// TwinCAT 3 PLC project Ligne
// ProgramVersion: 3.1.0.8
// libraries:
//   VisuElem3DPath, 3.5.4.0 (System)
//   VisuElemMeter, 3.5.4.0 (System)
//   VisuElems, 3.5.4.10 (System)
//   VisuElemsSpecialControls, 3.5.4.10 (System)
//   VisuElemsWinControls, 3.5.4.10 (System)
//   VisuElemTextEditor, 3.5.4.0 (System)
//   visuinputs, 3.5.4.0 (system)
//   VisuNativeControl, 3.5.4.0 (System)
//   Tc2_Standard, * (Beckhoff Automation GmbH)
//   Tc2_System, * (Beckhoff Automation GmbH)
//   Tc3_Interfaces, * (Beckhoff Automation GmbH)
//   Tc3_Module, * (Beckhoff Automation GmbH)
//   Maxon,1.0.0.0,Maxon Motor
//   Tc2_ControllerToolbox,3.4.1.0,Beckhoff Automation GmbH
//   Tc2_Utilities,3.3.8.0,Beckhoff Automation GmbH
// project tree:
//   DUTs/ FLAGS.TcDUT, FLOWMETER_CONTROL.TcDUT, FLOWMETER_SENSOR.TcDUT, FLOWMETER_VALUES.TcDUT, GAIN_SCHEDULED_PID.TcDUT, PRESSURE_SENSOR.TcDUT, PROG_STEPS.TcDUT, PUMP_PARAMS.TcDUT, SAFETY_IN.TcDUT, SAFETY_OUT.TcDUT
//   / GlobalTextList.TcGTLO, PlcTask.TcTTO, Visualization Manager.TcVMO (not stored)
//   GVLs/ Constant_Variables.TcGVL, Flag_Variables.TcGVL, IOs_Variables.TcGVL, PID_parameters.TcGVL
//   POUs/AIs/ AIS.TcPOU, ST45_TO_HMI.TcPOU
//   POUs/CONVOYER/ CONVEYOR.TcPOU, JIG.TcPOU
//   POUs/EAU/ VIDANGE_BALANCE_ST4.TcPOU, VIDANGE_BALANCE_ST5.TcPOU
//   POUs/EH/ EH_FLOMETER.TcPOU, EH_IEEE754_TO_REAL.TcPOU
//   POUs/Functions/ CONVERT_MASS_TO_FLOW.TcPOU, PRESSURE_REGULATOR.TcPOU
//   POUs/ GEMMA.TcPOU, MAIN.TcPOU
//   POUs/MAXON/ ST4_MOTOR.TcPOU, ST5_MOTOR.TcPOU, ST5_MOTOR_1.TcPOU
//   POUs/SAFETY/ SAFETY.TcPOU
//   POUs/STATIONS/ Q1.TcPOU, ST1_HT.TcPOU, ST2_ASPIRATION.TcPOU, ST3_ETANCHEITE.TcPOU, ST4_DEBIT_PETIT.TcPOU, ST5_GRAND_PETIT.TcPOU, ST7_SECHAGE.TcPOU, ST6_PMAX.TcPOU, ST8_IMPRESSION.TcPOU, ST9_DECHARGEMENT.TcPOU
//   POUs/WIKA/ WIKA_GET_VALUES.TcPOU
//   VISUs/ AIs.TcVIS, ST3.TcVIS, ST4.TcVIS, ST5.TcVIS, Visualization.TcVIS
// real-time tasks:
//   TASK PlcTask: cycle T#10ms, priority 20, ADS port 349
//   TASK Blinking: cycle T#450000us, priority 23, ADS port 351
//   TASK Slow_Tasks: cycle T#200000us, priority 22, ADS port 352
//   TASK TestOperator: cycle T#100000us, priority 21, ADS port 353
// I/O:
//   DEVICE Device 2 (EtherCAT), AmsNetId 10.10.10.31.3.1
//     Grande armoire [EK1100 EtherCAT Coupler (2A E-Bus)]
//       Term 51 (EL1002) [EL1002 2Ch. Dig. Input 24V, 3ms]
//       Term 52 (EL1002) [EL1002 2Ch. Dig. Input 24V, 3ms]
//       Term 53 (EL1002) [EL1002 2Ch. Dig. Input 24V, 3ms]
//       Term 54 (EL1002) [EL1002 2Ch. Dig. Input 24V, 3ms]
//       Term 55 (EL1002) [EL1002 2Ch. Dig. Input 24V, 3ms]
//       Term 56 (EL1002) [EL1002 2Ch. Dig. Input 24V, 3ms]
//       Term 57 (EL1002) [EL1002 2Ch. Dig. Input 24V, 3ms]
//       Term 58 (EL1002) [EL1002 2Ch. Dig. Input 24V, 3ms]
//       Term 59 (EL1002) [EL1002 2Ch. Dig. Input 24V, 3ms]
//       Term 60 (EL1002) [EL1002 2Ch. Dig. Input 24V, 3ms]
//       Term 61 (EL1002) [EL1002 2Ch. Dig. Input 24V, 3ms]
//       Term 62 (EL1002) [EL1002 2Ch. Dig. Input 24V, 3ms]
//       Term 63 (EL1002) [EL1002 2Ch. Dig. Input 24V, 3ms]
//       Term 64 (EL1002) [EL1002 2Ch. Dig. Input 24V, 3ms]
//       Term 65 (EL1002) [EL1002 2Ch. Dig. Input 24V, 3ms]
//       Term 66 (EL1002) [EL1002 2Ch. Dig. Input 24V, 3ms]
//       Term 67 (EL1002) [EL1002 2Ch. Dig. Input 24V, 3ms]
//       Term 68 (EL1002) [EL1002 2Ch. Dig. Input 24V, 3ms]
//       Term 32 (EL3064) [EL3064 4Ch. Ana. Input 0-10V]
//       Term 70 (EL1002) [EL1002 2Ch. Dig. Input 24V, 3ms]
//       Term 71 (EL9410) [EL9410 E-Bus Power Supplier  (Diagnostics)]
//       Term 72 (EL2002) [EL2002 2Ch. Dig. Output 24V, 0.5A]
//       Term 73 (EL2002) [EL2002 2Ch. Dig. Output 24V, 0.5A]
//       Term 74 (EL2002) [EL2002 2Ch. Dig. Output 24V, 0.5A]
//       Term 75 (EL2002) [EL2002 2Ch. Dig. Output 24V, 0.5A]
//       Term 76 (EL2002) [EL2002 2Ch. Dig. Output 24V, 0.5A]
//       Term 77 (EL2002) [EL2002 2Ch. Dig. Output 24V, 0.5A]
//       Term 78 (EL2002) [EL2002 2Ch. Dig. Output 24V, 0.5A]
//       Term 79 (EL2002) [EL2002 2Ch. Dig. Output 24V, 0.5A]
//       Term 80 (EL1512) [EL1512 2Ch. +/- Counter 24V, 1kHz]
//       Term 81 (EL2622) [EL2622 2Ch. Relay Output, NO (230V AC / 30V DC)]
//       Term 82 (EL2622) [EL2622 2Ch. Relay Output, NO (230V AC / 30V DC)]
//       Term 83 (EL2622) [EL2622 2Ch. Relay Output, NO (230V AC / 30V DC)]
//       Term 84 (EL2622) [EL2622 2Ch. Relay Output, NO (230V AC / 30V DC)]
//       Term 85 (EL2622) [EL2622 2Ch. Relay Output, NO (230V AC / 30V DC)]
//       Term 86 (EL2622) [EL2622 2Ch. Relay Output, NO (230V AC / 30V DC)]
//       Term 87 (EL3681) [EL3681 Digital multimeter terminal]
//       Term 88 (EL3681) [EL3681 Digital multimeter terminal]
//       Term 11 (EL2904) [EL2904, 4 Ch. Safety Output 24V, 0.5A, TwinSAFE]
//         modules: Module 1 (FSOES), Module 2 (DO)
//       Term 89 (EL6751) [EL6751 CANopen Master]
//       Term 90 (EL6751) [EL6751 CANopen Master]
//       Term 117 (EL9011) [EL9011 End Terminal]
//     Petite armoire [EK1100 EtherCAT Coupler (2A E-Bus)]
//       Term 92 (EL1002) [EL1002 2Ch. Dig. Input 24V, 3ms]
//       Term 93 (EL1002) [EL1002 2Ch. Dig. Input 24V, 3ms]
//       Term 94 (EL1002) [EL1002 2Ch. Dig. Input 24V, 3ms]
//       Term 95 (EL1002) [EL1002 2Ch. Dig. Input 24V, 3ms]
//       Term 96 (EL1002) [EL1002 2Ch. Dig. Input 24V, 3ms]
//       Term 97 (EL1002) [EL1002 2Ch. Dig. Input 24V, 3ms]
//       Term 98 (EL1002) [EL1002 2Ch. Dig. Input 24V, 3ms]
//       Term 99 (EL1002) [EL1002 2Ch. Dig. Input 24V, 3ms]
//       Term 100 (EL1002) [EL1002 2Ch. Dig. Input 24V, 3ms]
//       Term 101 (EL1002) [EL1002 2Ch. Dig. Input 24V, 3ms]
//       Term 102 (EL1002) [EL1002 2Ch. Dig. Input 24V, 3ms]
//       Term 103 (EL1002) [EL1002 2Ch. Dig. Input 24V, 3ms]
//       Term 104 (EL2002) [EL2002 2Ch. Dig. Output 24V, 0.5A]
//       Term 105 (EL2002) [EL2002 2Ch. Dig. Output 24V, 0.5A]
//       Term 106 (EL2002) [EL2002 2Ch. Dig. Output 24V, 0.5A]
//       Term 107 (EL2002) [EL2002 2Ch. Dig. Output 24V, 0.5A]
//       Term 149 (EL1008) [EL1008 8Ch. Dig. Input 24V, 3ms]
//       Term 150 (EL2008) [EL2008 8Ch. Dig. Output 24V, 0.5A]
//       Term 108 (EL3051) [EL3051 1Ch. Ana. Input 4-20mA]
//       Term 109 (EL9512) [EL9512 Power supply terminal 12V]
//       Term 110 (EL3356-0010) [EL3356-0010 1Ch. Ana. Input Resistor Bridge Terminal, 24bit, High Precision]
//       Term 111 (EL9512) [EL9512 Power supply terminal 12V]
//       Term 112 (EL3356-0010) [EL3356-0010 1Ch. Ana. Input Resistor Bridge Terminal, 24bit, High Precision]
//       Term 113 (EL6900) [EL6900, TwinSAFE PLC]
//       Term 114 (EL1904) [EL1904, 4 Ch. Safety Input 24V, TwinSAFE]
//         modules: Module 1 (FSOES)
//       Term 115 (EL1904) [EL1904, 4 Ch. Safety Input 24V, TwinSAFE]
//         modules: Module 1 (FSOES)
//       Term 116 (EL6731) [EL6731 PROFIBUS DP Master]
//       Term 118 (EL9011) [EL9011 End Terminal]
//     Box Etanchetie (EX260-SEC1) [EX260-SEC1 EtherCAT SI Unit (32DO_PNP) Rev1.2]
//     Box Debit (EX260-SEC1) [EX260-SEC1 EtherCAT SI Unit (32DO_PNP) Rev1.2]
//     Box Imprimante (EX260-SEC1) [EX260-SEC1 EtherCAT SI Unit (32DO_PNP) Rev1.2]
//   DEVICE Device 3 (EL6751), AmsNetId 10.10.10.31.4.1
//     Moteur Q1 (EPOS) (disabled)
//   DEVICE Device 4 (EL6751), AmsNetId 10.10.10.31.5.1
//     Moteur Q2 (EPOS) (disabled)
//   DEVICE Device 1 (EL6731), AmsNetId 10.10.10.31.2.1
//     Pressure Sensor 2P1 // Vendor: WIKA Revision: Rev 0.2
//     Pressure Sensor 4P2 // Vendor: WIKA Revision: Rev 0.2
//     Pressure Sensor 5P1 // Vendor: WIKA Revision: Rev 0.2
//     Pressure Sensor 5P2 // Vendor: WIKA Revision: Rev 0.2
//     Pressure Sensor 6P1 // Vendor: WIKA Revision: Rev 0.2
//     Pressure Sensor 4P1 // Vendor: WIKA Revision: Rev 0.2
// variable links:
//   Device 2 (EtherCAT) <-> Device 2 (EtherCAT)/Petite armoire/Term 113 (EL6900)
//     Grande armoire/Term 11 (EL2904)/Module 1 (FSOES)/RxPDO/FSOE <-> ConnectionInputs/Message_5 TxPDO
//     Grande armoire/Term 11 (EL2904)/Module 1 (FSOES)/TxPDO/FSOE <-> ConnectionOutputs/Message_5 RxPDO
//     Petite armoire/Term 114 (EL1904)/Module 1 (FSOES)/RxPDO/FSOE <-> ConnectionInputs/Message_24 TxPDO
//     Petite armoire/Term 114 (EL1904)/Module 1 (FSOES)/TxPDO/FSOE <-> ConnectionOutputs/Message_24 RxPDO
//     Petite armoire/Term 115 (EL1904)/Module 1 (FSOES)/TxPDO/FSOE <-> ConnectionOutputs/Message_4 RxPDO
//   Device 2 (EtherCAT) <-> Device 2 (EtherCAT)/Petite armoire/Term 115 (EL1904)
//     Petite armoire/Term 113 (EL6900)/ConnectionInputs/Message_4 TxPDO <-> Module 1 (FSOES)/RxPDO/FSOE
//   Ligne/Ligne Instance <-> Device 1 (EL6731)/Pressure Sensor 2P1
//     PlcTask Inputs/.ST2_2P1/VALUE <-> 8 Byte In, 3 Byte Out/Inputs/8 Byte In, 3 Byte Out_0_0
//   Ligne/Ligne Instance <-> Device 1 (EL6731)/Pressure Sensor 4P1
//     PlcTask Inputs/.ST4_4P1/VALUE <-> 8 Byte In, 3 Byte Out/Inputs/8 Byte In, 3 Byte Out_0_0
//   Ligne/Ligne Instance <-> Device 1 (EL6731)/Pressure Sensor 4P2
//     PlcTask Inputs/.ST4_4P2/VALUE <-> 8 Byte In, 3 Byte Out/Inputs/8 Byte In, 3 Byte Out_0_0
//   Ligne/Ligne Instance <-> Device 1 (EL6731)/Pressure Sensor 5P1
//     PlcTask Inputs/.ST5_5P1/VALUE <-> 8 Byte In, 3 Byte Out/Inputs/8 Byte In, 3 Byte Out_0_0
//   Ligne/Ligne Instance <-> Device 1 (EL6731)/Pressure Sensor 5P2
//     PlcTask Inputs/.ST5_5P2/VALUE <-> 8 Byte In, 3 Byte Out/Inputs/8 Byte In, 3 Byte Out_0_0
//   Ligne/Ligne Instance <-> Device 1 (EL6731)/Pressure Sensor 6P1
//     PlcTask Inputs/.ST6_6P1/VALUE <-> 8 Byte In, 3 Byte Out/Inputs/8 Byte In, 3 Byte Out_0_0
//   Ligne/Ligne Instance <-> Device 2 (EtherCAT)/Box Debit (EX260-SEC1)
//     PlcTask Outputs/.ST4_4V1 <-> Byte 0/Output
//     PlcTask Outputs/.ST5_5V2 <-> Byte 1/Output
//     PlcTask Outputs/.ST6_6V4 <-> Byte 2/Output
//     PlcTask Outputs/.ST4_4V2 <-> Byte 0/Output @bit 1
//     PlcTask Outputs/.ST4_4V3 <-> Byte 0/Output @bit 2
//     PlcTask Outputs/.ST4_4V4 <-> Byte 0/Output @bit 3
//     PlcTask Outputs/.ST4_4V5 <-> Byte 0/Output @bit 4
//     PlcTask Outputs/.ST4_4V6 <-> Byte 0/Output @bit 5
//     PlcTask Outputs/.ST4_4V7 <-> Byte 0/Output @bit 6
//     PlcTask Outputs/.ST5_5V1 <-> Byte 0/Output @bit 7
//     PlcTask Outputs/.ST5_5V3 <-> Byte 1/Output @bit 1
//     PlcTask Outputs/.ST5_5V4 <-> Byte 1/Output @bit 2
//     PlcTask Outputs/.ST5_5V5 <-> Byte 1/Output @bit 3
//     PlcTask Outputs/.ST5_5V6 <-> Byte 1/Output @bit 4
//     PlcTask Outputs/.ST6_6V1 <-> Byte 1/Output @bit 5
//     PlcTask Outputs/.ST6_6V2 <-> Byte 1/Output @bit 6
//     PlcTask Outputs/.ST6_6V3 <-> Byte 1/Output @bit 7
//     PlcTask Outputs/.ST6_6V5 <-> Byte 2/Output @bit 1
//     PlcTask Outputs/.ST6_6V6 <-> Byte 2/Output @bit 2
//     PlcTask Outputs/.ST6_6V7 <-> Byte 2/Output @bit 3
//   Ligne/Ligne Instance <-> Device 2 (EtherCAT)/Box Etanchetie (EX260-SEC1)
//     PlcTask Outputs/.ST10_10V1 <-> Byte 0/Output
//     PlcTask Outputs/.ST2_2V2 <-> Byte 1/Output
//     PlcTask Outputs/.ST3_3V3 <-> Byte 2/Output
//     PlcTask Outputs/.ST10_10V2 <-> Byte 0/Output @bit 1
//     PlcTask Outputs/.ST1_1V1 <-> Byte 0/Output @bit 2
//     PlcTask Outputs/.ST1_1V2 <-> Byte 0/Output @bit 3
//     PlcTask Outputs/.ST1_1V3 <-> Byte 0/Output @bit 4
//     PlcTask Outputs/.ST1_1V4 <-> Byte 0/Output @bit 5
//     PlcTask Outputs/.ST1_1V5 <-> Byte 0/Output @bit 6
//     PlcTask Outputs/.ST2_2V1 <-> Byte 0/Output @bit 7
//     PlcTask Outputs/.ST2_2V3 <-> Byte 1/Output @bit 1
//     PlcTask Outputs/.ST2_2V4 <-> Byte 1/Output @bit 2
//     PlcTask Outputs/.ST2_2V5 <-> Byte 1/Output @bit 3
//     PlcTask Outputs/.ST2_2V6 <-> Byte 1/Output @bit 4
//     PlcTask Outputs/.ST2_2V7 <-> Byte 1/Output @bit 5
//     PlcTask Outputs/.ST3_3V1 <-> Byte 1/Output @bit 6
//     PlcTask Outputs/.ST3_3V2 <-> Byte 1/Output @bit 7
//     PlcTask Outputs/.ST3_3V4 <-> Byte 2/Output @bit 1
//     PlcTask Outputs/.ST3_3V5 <-> Byte 2/Output @bit 2
//     PlcTask Outputs/.ST3_3V7 <-> Byte 2/Output @bit 3
//   Ligne/Ligne Instance <-> Device 2 (EtherCAT)/Box Imprimante (EX260-SEC1)
//     PlcTask Outputs/.ST7_7V1 <-> Byte 0/Output @bit 1
//     PlcTask Outputs/.ST7_7V2 <-> Byte 0/Output @bit 2
//     PlcTask Outputs/.ST7_7V3 <-> Byte 0/Output @bit 3
//     PlcTask Outputs/.ST7_7V4 <-> Byte 0/Output @bit 4
//     PlcTask Outputs/.ST7_7V5 <-> Byte 0/Output @bit 5
//     PlcTask Outputs/.ST7_7V6 <-> Byte 0/Output @bit 6
//     PlcTask Outputs/.ST7_7V7 <-> Byte 0/Output @bit 7
//     PlcTask Outputs/.ST8_8V2 <-> Byte 1/Output @bit 1
//     PlcTask Outputs/.ST8_8V3 <-> Byte 1/Output @bit 2
//     PlcTask Outputs/.ST8_8V4 <-> Byte 1/Output @bit 3
//     PlcTask Outputs/.ST9_9V1 <-> Byte 1/Output @bit 4
//     PlcTask Outputs/.ST9_9V2 <-> Byte 1/Output @bit 5
//     PlcTask Outputs/.ST9_9V3 <-> Byte 1/Output @bit 6
//     PlcTask Outputs/.ST9_9V6 <-> Byte 2/Output @bit 3
//     PlcTask Outputs/.ST9_9V7 <-> Byte 2/Output @bit 4
//     PlcTask Outputs/.ST7_RESERVE <-> Byte 0/Output
//     PlcTask Outputs/.ST8_8V1 <-> Byte 1/Output
//     PlcTask Outputs/.ST9_9V4A <-> Byte 1/Output @bit 7
//     PlcTask Outputs/.ST9_9V5A <-> Byte 2/Output @bit 1
//     PlcTask Outputs/.ST9_9V4B <-> Byte 2/Output
//     PlcTask Outputs/.ST9_9V5B <-> Byte 2/Output @bit 2
//   Ligne/Ligne Instance <-> Device 2 (EtherCAT)/Grande armoire/Term 32 (EL3064)
//     PlcTask Inputs/.ST3_3P2 <-> AI Standard Channel 4/Value
//     PlcTask Inputs/.ST5_Niveau_Reservoir <-> AI Standard Channel 3/Value
//   Ligne/Ligne Instance <-> Device 2 (EtherCAT)/Grande armoire/Term 51 (EL1002)
//     PlcTask Inputs/.ST4_4B1 <-> Channel 1/4B1
//     PlcTask Inputs/.ST4_4B2 <-> Channel 2/4B2
//   Ligne/Ligne Instance <-> Device 2 (EtherCAT)/Grande armoire/Term 52 (EL1002)
//     PlcTask Inputs/.ST4_4B4 <-> Channel 1/4B4
//     PlcTask Inputs/.ST4_4B5 <-> Channel 2/4B5
//   Ligne/Ligne Instance <-> Device 2 (EtherCAT)/Grande armoire/Term 53 (EL1002)
//     PlcTask Inputs/.ST4_4B6 <-> Channel 1/4B6
//     PlcTask Inputs/.ST4_4B7 <-> Channel 2/4B7
//   Ligne/Ligne Instance <-> Device 2 (EtherCAT)/Grande armoire/Term 54 (EL1002)
//     PlcTask Inputs/.ST5_5B1 <-> Channel 1/5B1
//     PlcTask Inputs/.ST5_5B2 <-> Channel 2/5B2
//   Ligne/Ligne Instance <-> Device 2 (EtherCAT)/Grande armoire/Term 55 (EL1002)
//     PlcTask Inputs/.ST5_5B4 <-> Channel 1/5B4
//     PlcTask Inputs/.ST5_5B5 <-> Channel 2/5B5
//   Ligne/Ligne Instance <-> Device 2 (EtherCAT)/Grande armoire/Term 56 (EL1002)
//     PlcTask Inputs/.ST5_5B6 <-> Channel 1/5B6
//   Ligne/Ligne Instance <-> Device 2 (EtherCAT)/Grande armoire/Term 57 (EL1002)
//     PlcTask Inputs/.ST6_6B1 <-> Channel 1/6B1
//     PlcTask Inputs/.ST6_6B2 <-> Channel 2/6B2
//   Ligne/Ligne Instance <-> Device 2 (EtherCAT)/Grande armoire/Term 58 (EL1002)
//     PlcTask Inputs/.ST6_6B4 <-> Channel 1/6B4
//     PlcTask Inputs/.ST6_6B5 <-> Channel 2/6B5
//   Ligne/Ligne Instance <-> Device 2 (EtherCAT)/Grande armoire/Term 59 (EL1002)
//     PlcTask Inputs/.ST6_6B6 <-> Channel 1/6B6
//     PlcTask Inputs/.ST6_6B7 <-> Channel 2/6B7
//   Ligne/Ligne Instance <-> Device 2 (EtherCAT)/Grande armoire/Term 60 (EL1002)
//     PlcTask Inputs/.ST7_7B1 <-> Channel 1/7B1
//     PlcTask Inputs/.ST7_7B2 <-> Channel 2/7B2
//   Ligne/Ligne Instance <-> Device 2 (EtherCAT)/Grande armoire/Term 61 (EL1002)
//     PlcTask Inputs/.ST7_7B4 <-> Channel 1/7B4
//     PlcTask Inputs/.ST7_7B5 <-> Channel 2/7B5
//   Ligne/Ligne Instance <-> Device 2 (EtherCAT)/Grande armoire/Term 62 (EL1002)
//     PlcTask Inputs/.ST7_7B6 <-> Channel 1/7B6
//     PlcTask Inputs/.ST7_7B7 <-> Channel 2/7B7
//   Ligne/Ligne Instance <-> Device 2 (EtherCAT)/Grande armoire/Term 63 (EL1002)
//     PlcTask Inputs/.ST8_8B1 <-> Channel 1/8B1
//     PlcTask Inputs/.ST8_8B2 <-> Channel 2/8B2
//   Ligne/Ligne Instance <-> Device 2 (EtherCAT)/Grande armoire/Term 64 (EL1002)
//     PlcTask Inputs/.ST9_9B1 <-> Channel 1/9B1
//     PlcTask Inputs/.ST9_9B2 <-> Channel 2/9B2
//   Ligne/Ligne Instance <-> Device 2 (EtherCAT)/Grande armoire/Term 65 (EL1002)
//     PlcTask Inputs/.ST9_9B4 <-> Channel 1/9B4
//     PlcTask Inputs/.ST9_9B41 <-> Channel 2/9B4.1
//   Ligne/Ligne Instance <-> Device 2 (EtherCAT)/Grande armoire/Term 66 (EL1002)
//     PlcTask Inputs/.ST9_9B5 <-> Channel 1/9B5
//     PlcTask Inputs/.ST9_9B51 <-> Channel 2/9B5.1
//   Ligne/Ligne Instance <-> Device 2 (EtherCAT)/Grande armoire/Term 67 (EL1002)
//     PlcTask Inputs/.ST9_9B6 <-> Channel 1/9B6
//     PlcTask Inputs/.ST9_9B7 <-> Channel 2/9B7
//   Ligne/Ligne Instance <-> Device 2 (EtherCAT)/Grande armoire/Term 68 (EL1002)
//     PlcTask Inputs/.ST9_9B61 <-> Channel 2/9B6.1
//   Ligne/Ligne Instance <-> Device 2 (EtherCAT)/Grande armoire/Term 72 (EL2002)
//     PlcTask Outputs/.ST4_4V10 <-> Channel 1/4V10
//     PlcTask Outputs/.ST4_4V12 <-> Channel 2/4V12
//   Ligne/Ligne Instance <-> Device 2 (EtherCAT)/Grande armoire/Term 73 (EL2002)
//     PlcTask Outputs/.ST4_4V13 <-> Channel 1/4V13
//   Ligne/Ligne Instance <-> Device 2 (EtherCAT)/Grande armoire/Term 74 (EL2002)
//     PlcTask Outputs/.ST5_5V10 <-> Channel 1/5V10
//     PlcTask Outputs/.ST5_5V12 <-> Channel 2/5V12
//   Ligne/Ligne Instance <-> Device 2 (EtherCAT)/Grande armoire/Term 75 (EL2002)
//     PlcTask Outputs/.ST5_5V13 <-> Channel 1/5V13
//     PlcTask Outputs/.ST5_5V14 <-> Channel 2/5V14
//   Ligne/Ligne Instance <-> Device 2 (EtherCAT)/Grande armoire/Term 76 (EL2002)
//     PlcTask Outputs/.ST5_5V15 <-> Channel 1/5V15
//     PlcTask Outputs/.ST5_5V16 <-> Channel 2/5V16
//   Ligne/Ligne Instance <-> Device 2 (EtherCAT)/Grande armoire/Term 77 (EL2002)
//     PlcTask Outputs/.ST6_6V10 <-> Channel 1/6V10
//     PlcTask Outputs/.ST6_6V11 <-> Channel 2/6V11
//   Ligne/Ligne Instance <-> Device 2 (EtherCAT)/Grande armoire/Term 78 (EL2002)
//     PlcTask Outputs/.GEN_CONVOYEUR <-> Channel 1/K2
//   Ligne/Ligne Instance <-> Device 2 (EtherCAT)/Grande armoire/Term 79 (EL2002)
//     PlcTask Outputs/.ST7_7V10 <-> Channel 1/7V10
//   Ligne/Ligne Instance <-> Device 2 (EtherCAT)/Grande armoire/Term 81 (EL2622)
//     PlcTask Outputs/.ST2_POWER <-> Channel 1/2M1L
//     PlcTask Outputs/.ST2_POWER <-> Channel 2/2M1N
//   Ligne/Ligne Instance <-> Device 2 (EtherCAT)/Grande armoire/Term 82 (EL2622)
//     PlcTask Outputs/.ST4_POWER <-> Channel 1/4M1L
//     PlcTask Outputs/.ST4_POWER <-> Channel 2/4M1N
//   Ligne/Ligne Instance <-> Device 2 (EtherCAT)/Grande armoire/Term 83 (EL2622)
//     PlcTask Outputs/.ST5_POWER <-> Channel 1/5M1L
//     PlcTask Outputs/.ST5_POWER <-> Channel 2/5M1N
//   Ligne/Ligne Instance <-> Device 2 (EtherCAT)/Grande armoire/Term 84 (EL2622)
//     PlcTask Outputs/.ST6_POWER <-> Channel 1/6M1L
//     PlcTask Outputs/.ST6_POWER <-> Channel 2/6M1N
//   Ligne/Ligne Instance <-> Device 2 (EtherCAT)/Grande armoire/Term 85 (EL2622)
//     PlcTask Outputs/.ST7_POWER <-> Channel 1/7M1L
//     PlcTask Outputs/.ST7_POWER <-> Channel 2/7M1N
//   Ligne/Ligne Instance <-> Device 2 (EtherCAT)/Grande armoire/Term 86 (EL2622)
//     PlcTask Outputs/.ST4_VIDANGE <-> Channel 1/4M2
//     PlcTask Outputs/.ST5_VIDANGE <-> Channel 2/5M2
//   Ligne/Ligne Instance <-> Device 2 (EtherCAT)/Grande armoire/Term 87 (EL3681)
//     PlcTask Inputs/.ST4_Multimeter_value <-> SAI Inputs/Value
//     PlcTask Outputs/.ST4_Multimeter_mode <-> SAI Range/Control/Mode
//     PlcTask Outputs/.ST4_Multimeter_range <-> SAI Range/Control/Range
//   Ligne/Ligne Instance <-> Device 2 (EtherCAT)/Grande armoire/Term 88 (EL3681)
//     PlcTask Inputs/.ST5_Multimeter_value <-> SAI Inputs/Value
//     PlcTask Outputs/.ST5_Multimeter_mode <-> SAI Range/Control/Mode
//     PlcTask Outputs/.ST5_Multimeter_range <-> SAI Range/Control/Range
//   Ligne/Ligne Instance <-> Device 2 (EtherCAT)/Petite armoire/Term 100 (EL1002)
//     PlcTask Inputs/.GEN_PRESENCE_POMPE <-> Channel 1/Présence pompe
//   Ligne/Ligne Instance <-> Device 2 (EtherCAT)/Petite armoire/Term 101 (EL1002)
//     PlcTask Inputs/.ST4_DIGMESA <-> Channel 1/Input
//   Ligne/Ligne Instance <-> Device 2 (EtherCAT)/Petite armoire/Term 102 (EL1002)
//     PlcTask Inputs/.ST10_OPERATEUR1_START <-> Channel 1/S1
//     PlcTask Inputs/.ST10_OPERATEUR2_START <-> Channel 2/S2
//   Ligne/Ligne Instance <-> Device 2 (EtherCAT)/Petite armoire/Term 103 (EL1002)
//     PlcTask Inputs/.ST10_10B1 <-> Channel 1/10B1
//     PlcTask Inputs/.ST10_10B2 <-> Channel 2/10B2
//   Ligne/Ligne Instance <-> Device 2 (EtherCAT)/Petite armoire/Term 104 (EL2002)
//     PlcTask Outputs/.ST3_3V10 <-> Channel 1/3V10
//     PlcTask Outputs/.ST3_3V11 <-> Channel 2/3V11
//   Ligne/Ligne Instance <-> Device 2 (EtherCAT)/Petite armoire/Term 105 (EL2002)
//     PlcTask Outputs/.ST2_2V8 <-> Channel 2/2V8
//     PlcTask Outputs/.ST3_3V12 <-> Channel 1/3V12
//   Ligne/Ligne Instance <-> Device 2 (EtherCAT)/Petite armoire/Term 106 (EL2002)
//     PlcTask Outputs/.GEN_1V1 <-> Channel 1/0V1
//   Ligne/Ligne Instance <-> Device 2 (EtherCAT)/Petite armoire/Term 108 (EL3051)
//     PlcTask Inputs/.ST3_3P1 <-> AI Standard/3P1
//   Ligne/Ligne Instance <-> Device 2 (EtherCAT)/Petite armoire/Term 110 (EL3356-0010)
//     PlcTask Inputs/.ST4_POIDS <-> RMB Value (Real)/4U1
//   Ligne/Ligne Instance <-> Device 2 (EtherCAT)/Petite armoire/Term 112 (EL3356-0010)
//     PlcTask Inputs/.ST5_POIDS <-> RMB Value (Real)/5U1
//   Ligne/Ligne Instance <-> Device 2 (EtherCAT)/Petite armoire/Term 113 (EL6900)
//     PlcTask Inputs/.SAFETY_IN/NOT_AUS_State <-> Function Block Info Data/TwinSafeGroup2.Network1.FBEstop1 Info Data/State
//     PlcTask Outputs/.SAFETY_OUT/NOT_AUS_ErrAck <-> StandardOutputs/Standard In Var 9
//     PlcTask Outputs/.SAFETY_OUT/NOT_AUS_RESET <-> StandardOutputs/Standard In Var 10
//     PlcTask Outputs/.SAFETY_OUT/NOT_AUS_RUN <-> StandardOutputs/Standard In Var 8
//   Ligne/Ligne Instance <-> Device 2 (EtherCAT)/Petite armoire/Term 149 (EL1008)
//     PlcTask Inputs/.ST1_HT_CTRLOUT <-> Channel 1/HT_CTRLout
//     PlcTask Inputs/.ST1_HT_EOT <-> Channel 2/HT_EOT
//     PlcTask Inputs/.ST1_HT_ERROR <-> Channel 5/ERROR
//     PlcTask Inputs/.ST1_HT_FAIL <-> Channel 4/HT_FAIL
//     PlcTask Inputs/.ST1_HT_PASS <-> Channel 3/HT_PASS
//   Ligne/Ligne Instance <-> Device 2 (EtherCAT)/Petite armoire/Term 150 (EL2008)
//     PlcTask Outputs/.ST1_HT_CTRLIN <-> Channel 1/HT_CTRLIN
//     PlcTask Outputs/.ST1_HT_MES_DCH <-> Channel 6/HT_MES_DCH
//     PlcTask Outputs/.ST1_HT_N0 <-> Channel 3/HT_N0
//     PlcTask Outputs/.ST1_HT_N1 <-> Channel 4/HT_N1
//     PlcTask Outputs/.ST1_HT_N2 <-> Channel 5/HT_N2
//     PlcTask Outputs/.ST1_HT_TYPW <-> Channel 2/HT_TYPE
//   Ligne/Ligne Instance <-> Device 2 (EtherCAT)/Petite armoire/Term 92 (EL1002)
//     PlcTask Inputs/.ST1_1B1 <-> Channel 1/1B1
//     PlcTask Inputs/.ST1_1B2 <-> Channel 2/1B2
//   Ligne/Ligne Instance <-> Device 2 (EtherCAT)/Petite armoire/Term 93 (EL1002)
//     PlcTask Inputs/.ST1_1B4 <-> Channel 1/1B4
//     PlcTask Inputs/.ST1_1B5 <-> Channel 2/1B5
//   Ligne/Ligne Instance <-> Device 2 (EtherCAT)/Petite armoire/Term 94 (EL1002)
//     PlcTask Inputs/.ST2_2B1 <-> Channel 1/2B1
//     PlcTask Inputs/.ST2_2B2 <-> Channel 2/2B2
//   Ligne/Ligne Instance <-> Device 2 (EtherCAT)/Petite armoire/Term 95 (EL1002)
//     PlcTask Inputs/.ST2_2B4 <-> Channel 1/2B4
//     PlcTask Inputs/.ST2_2B5 <-> Channel 2/2B5
//   Ligne/Ligne Instance <-> Device 2 (EtherCAT)/Petite armoire/Term 96 (EL1002)
//     PlcTask Inputs/.ST2_2B6 <-> Channel 1/2B6
//     PlcTask Inputs/.ST2_2B7 <-> Channel 2/2B7
//   Ligne/Ligne Instance <-> Device 2 (EtherCAT)/Petite armoire/Term 97 (EL1002)
//     PlcTask Inputs/.ST3_3B1 <-> Channel 1/3B1
//     PlcTask Inputs/.ST3_3B2 <-> Channel 2/3B2
//   Ligne/Ligne Instance <-> Device 2 (EtherCAT)/Petite armoire/Term 98 (EL1002)
//     PlcTask Inputs/.ST3_3B4 <-> Channel 1/3B4
//     PlcTask Inputs/.ST3_3B5 <-> Channel 2/3B5
//   Ligne/Ligne Instance <-> Device 2 (EtherCAT)/Petite armoire/Term 99 (EL1002)
//     PlcTask Inputs/.GEN_0B1 <-> Channel 2/0B1
//     PlcTask Inputs/.ST3_3B7 <-> Channel 1/3B7

CONFIGURATION Ligne
    RESOURCE PLC ON TwinCAT3
        TASK PlcTask(INTERVAL := T#10ms, PRIORITY := 20);
        PROGRAM MAIN WITH PlcTask : MAIN;
    END_RESOURCE
END_CONFIGURATION

// ---- DUTs/FLAGS.TcDUT
TYPE FLAGS :
STRUCT

	INIT_OK:BOOL;
	SAFETY_OK:BOOL;
	MANUAL:BOOL;
	AUTO:BOOL;
	
	DEBUG_OPERATOR:BOOL;
	
	ST1_JIG_STATUS: BOOL;
	ST1_RELEASE_CARRIER:BOOL;
	ST2_JIG_STATUS: BOOL;
	ST2_RELEASE_CARRIER:BOOL;
	ST3_JIG_STATUS: BOOL;
	ST3_RELEASE_CARRIER:BOOL;
	ST4_JIG_STATUS: BOOL;
	ST4_RELEASE_CARRIER:BOOL;
	ST5_JIG_STATUS: BOOL;
	ST5_RELEASE_CARRIER:BOOL;
	ST6_JIG_STATUS: BOOL;
	ST6_RELEASE_CARRIER:BOOL;
	ST7_JIG_STATUS: BOOL;
	ST7_RELEASE_CARRIER:BOOL;
	ST8_JIG_STATUS: BOOL;
	ST8_RELEASE_CARRIER:BOOL;
	ST9_JIG_STATUS: BOOL;
	ST9_RELEASE_CARRIER:BOOL;

	
	DOORS_OPEN:BOOL;
	F2_END:BOOL;
	GEMMA: STRING;
	
	MOTOR_ST4_INIT_OK:BOOL;
	MOTOR_ST4_POSITION:DINT;
	MOTOR_ST4_ACTUAL_POSITION:DINT;
	MOTOR_ST5_INIT_OK:BOOL;
	MOTOR_ST5_POSITION:DINT;
	MOTOR_ST5_ACTUAL_POSITION:DINT;



END_STRUCT
END_TYPE

// ---- DUTs/FLOWMETER_CONTROL.TcDUT
TYPE FLOWMETER_CONTROL :
STRUCT

	SET_TOT: USINT;
	SET_MODE: USINT;

END_STRUCT
END_TYPE

// ---- DUTs/FLOWMETER_SENSOR.TcDUT

(************************************************************************************************
*
*Variables structure for E&H flowmeter PROMAS 83A
*
***********************************************************************************************)


TYPE FLOWMETER_SENSOR :
STRUCT

	A1 :ARRAY[0..4] OF USINT;
	A2 :ARRAY[0..4] OF USINT;
	A3 :ARRAY[0..4] OF USINT;
	A4 :ARRAY[0..4] OF USINT;
	A5 :ARRAY[0..4] OF USINT;
	A6 :ARRAY[0..4] OF USINT;
	TOT :ARRAY[0..4] OF USINT;

END_STRUCT
END_TYPE

// ---- DUTs/FLOWMETER_VALUES.TcDUT
TYPE FLOWMETER_VALUES :
STRUCT
	MassFlow:REAL;
	VolumeFlow:REAL;
	CorrectedVolueFLow:REAL;
	Density:REAL;
	ReferenceDensity:REAL;
	Temperature:REAL;
	TotalMass:REAL;
END_STRUCT
END_TYPE

// ---- DUTs/GAIN_SCHEDULED_PID.TcDUT
TYPE GAIN_SCHEDULED_PID :
STRUCT
	q			:REAL; 	(*gain scheduled parameter for which this PID is optimized*)
	Kp			:REAL;	(*constant for proportional part of the PID*)
	Ki			:REAL;	(*constant for integral part of the PID*)
	Kd			:REAL;	(*constant for derivative part of the PID*)
END_STRUCT
END_TYPE

// ---- DUTs/PRESSURE_SENSOR.TcDUT

(************************************************************************************************
*
*Variables structure for WIKA pressure sensor
*
***********************************************************************************************)

TYPE PRESSURE_SENSOR :
STRUCT

	VALUE :ARRAY [0..7] OF USINT;

END_STRUCT
END_TYPE

// ---- DUTs/PROG_STEPS.TcDUT
TYPE PROG_STEPS :
STRUCT

	ST1:INT;
	ST2:INT;
	ST3:INT;
	ST4:INT;
	ST5:INT;
	ST6:INT;
	ST7:INT;
	ST8:INT;
	ST9:INT;


END_STRUCT
END_TYPE

// ---- DUTs/PUMP_PARAMS.TcDUT
TYPE PUMP_PARAMS :
STRUCT
	
(* Général *******************************************************************************************************************)
	GEN_GRAND_DEBIT					:BOOL:=FALSE;		(*FALSE / ST4 petit débit     TRUE / ST5 grand débit*)
	GEN_BYPASS						:BOOL:=FALSE;		(*FALSE / N'utilise pas le contrôle du bypass      TRUE / Utilise le contrôle du by-pass*)
		
	
(* Station 1 Haute tension ***************************************************************************************************)
	ST1_HT_NO_PROG					:INT:=1;			(*Numéro de programme de l'appareil de test HT*)

(* Station 2 aspiration ******************************************************************************************************)
	ST2_CONTRE_PRESSION				:BOOL:=0;			(*Contre pression d'air TRUE: avec contre pression FALSE: sans contre pression*)
	ST2_TEMPS_POMPAGE				:TIME:= T#10S;		(*Temps d'amorcage *)
	ST2_TEMPS_MESURE				:TIME:= T#5S;		(*Temps de mesure *)
	ST2_TEMPS_MESURE_PERTE_PRESSION	:TIME:= T#2S;		(*Temps de mesure perte pression - PAS PROGRAMME *)
		
(* Station 3 étanchéité ******************************************************************************************************)
	ST3_TEMPS_MISE_SOUS_PRESSION	:TIME:= T#5S;		(*Temps de mise sous pression*)
	ST3_TEMPS_STABILISATION			:TIME:= T#10S;		(*Temps de stabilisation de la pression*)
	ST3_TEMPS_MESURE				:TIME:= T#15S;		(*Temps de mesure de la chutte de	 pression*)
	

(* Station 4-5 Débit *****************************************************************************************************)
	ST45_TEMPS_POMPAGE				:TIME:= T#10S;		(*Temps amorcage de la pompe *)
	ST45_TEMPS_MESURE_DEBIT_MAX		:TIME:= T#10S;		(*Temps de mesure de Qmax*)
	ST45_TEMPS_REGLAGE_PRESSION		:TIME:= T#30S;		(*Temps de réglage de la pression *)
	ST45_TEMPS_MESURE_DEBIT			:TIME:= T#10S;		(*Temps de mesure de Qtravail *)
	ST45_PRESSION_CONSIGNE			:REAL:= 7.0;		(*Presssion de consigne pour le débit de travail*)

(* Station 6 Pmax ************************************************************************************************************)	
	ST6_TEMPS_POMPAGE				:TIME:= T#10S;		(*Temps amorcage de la pompe *)
	ST6_TEMPS_MESURE				:TIME:= T#5S;		(*Temps de mesure de Pmax *)
	ST6_TEMPS_MESURE_PERTE_PRESSION	:TIME:= T#1S;		(*Temps de mesure perte de pression max - PAS PROGRAMME *)
	
(* Station 7 Sechage *********************************************************************************************************)
	ST7_TEMPS_SECHAGE				:TIME:= T#2S;		(*Temps séchage pompe station 7 *)
	
(* Station 9 Déchargement*****************************************************************************************************)
	ST9_BOBINE_A_FIL				:BOOL:=TRUE;		(*Si bobine à fil, utilise de vérin de débloquage des fils *)



END_STRUCT
END_TYPE

// ---- DUTs/SAFETY_IN.TcDUT
TYPE SAFETY_IN :
STRUCT

	NOT_AUS_State:USINT;

END_STRUCT
END_TYPE

// ---- DUTs/SAFETY_OUT.TcDUT
TYPE SAFETY_OUT :
STRUCT


	NOT_AUS_RUN:BOOL;
	NOT_AUS_ErrAck:BOOL;
	NOT_AUS_RESET:BOOL;

END_STRUCT
END_TYPE

// ---- GVLs/Constant_Variables.TcGVL
{attribute 'Tc2GvlVarNames'}
VAR_GLOBAL
	(********************
	*
	* Times
	*  
	************************)
	CARRIER_RELEASE_DELAY						:TIME:= T#600MS;			(*Temps de rentrée du vérin de blocage des vérins*)
	PULSE_RELEASE_JIG_OP						:TIME:= T#250MS;		(*Duration of the pulse to release a carrier on the Operators jig*)
	DELAY_EJECT_CARRIERS						:TIME:= T#5S;			(*Time for release all the carriers present in the tunel during the initialisation *)
	DELAY_START_AIR								:TIME:= T#2S;			(*Time to let air starting before starting convoyer *)

	TEMPS_VIDANGE_POMPE							:TIME:= T#5S;			(*Temps durant lequel on pompe de l'air pour vidanger la pompe*)
	TEMPS_VIDANGE_RESERVOIR						:TIME:= T#30S;			(*Temps durant lequel on continue de vider le réservoir d'eau pour être sur qu'il est vide*)
	
	TEMPS_SORTIE_VERIN							:TIME:= T#3S;			(*Temps durant lequel on pompe de l'air pour vidanger la pompe*)
	TEMPS_RENTREE_VERIN							:TIME:= T#1S;			(*Temps laissé au vérin pour rentrer avant que la palette soit libérée*)
	TEMPS_CHANGEMENT_PRESSION					:TIME:= T#4S;			(*Temps pour la mise sous pression du débit de travail avant réglage*)

	(********************
	*
	* Motor
	*
	************************)
	MOTOR_ST4_ADDRESS							:STRING:= '10.10.10.31.4.1';	(*Adresse moteur ST4*)
	MOTOR_ST5_ADDRESS							:STRING:= '10.10.10.31.5.1';	(*Adresse moteur ST5*)
	MOTOR_ST4_INITIAL_POS						:DINT:=25000;					(*Initial position of the motor*)
	MOTOR_ST4_POSITION_MAX						:DINT:=35000;					(*Butée soft du moteur*)
	MOTOR_ST5_INITIAL_POS						:DINT:=25000;					(*Initial position of the motor*)
	MOTOR_ST5_POSITION_MAX						:DINT:=35000;					(*Butée soft du moteur*)
	
	RESERVOIR_EAU_MAX							:INT:=5000;						(*Niveau haut du réservoir d'eau*)
	RESERVOIR_EAU_MIN							:INT:=14000;					(*Niveau bas du réservoir d'eau*)
	
	(********************
	*
	* Weigthing
	*
	************************)
	
	BALANCE_POIDS_LIMITE								:INT:=2000;

END_VAR

VAR_GLOBAL

	(********************
	*
	* Config
	*
	************************)

	PUMP_PARAMS 									: PUMP_PARAMS;		(*Paramètre de test qu viennent depuis Labview*)

	(********************
	*
	* Activation des Posages
	*
	************************)
	ST1_JIG_DISABLED							:BOOL:=FALSE;			(*Désactive le posage*)
	ST2_JIG_DISABLED							:BOOL:=FALSE;			(*Désactive le posage*)
	ST3_JIG_DISABLED							:BOOL:=FALSE;			(*Désactive le posage*)
	ST4_5_JIG_DISABLED							:BOOL:=FALSE;			(*Désactive les posages ST4 et ST5*)
	ST6_JIG_DISABLED							:BOOL:=FALSE;			(*Désactive le posage*)
	ST7_JIG_DISABLED							:BOOL:=FALSE;			(*Désactive le posage*)
	ST8_JIG_DISABLED							:BOOL:=FALSE;			(*Désactive le posage*)
	ST9_JIG_DISABLED							:BOOL:=FALSE;			(*Désactive le posage*)
	ST4_JIG_DISABLED							:BOOL;					(*via la variable GRAND_DEBIT*)
	ST5_JIG_DISABLED							:BOOL;					(*via la variable GRAND_DEBIT*)

END_VAR

// ---- GVLs/Flag_Variables.TcGVL
{attribute 'Tc2GvlVarNames'}
VAR_GLOBAL


	FLAGS 				AT%M*: FLAGS;


	SAFETY_IN 			AT%I*: SAFETY_IN;
	SAFETY_OUT 			AT%Q*: SAFETY_OUT;

	(*Visualisation des débits ST4*)
	QMAX_ARRAY: ARRAY[1..50] OF REAL;
	INDEX_QMAX_ARRAY :INT:=1;
	Q_ARRAY: ARRAY[1..50] OF REAL;
	INDEX_Q_ARRAY :INT:=1;
	
	QMAX5_ARRAY: ARRAY[1..50] OF REAL;
	INDEX_QMAX5_ARRAY :INT:=1;
	Q5_ARRAY: ARRAY[1..50] OF REAL;
	INDEX_Q5_ARRAY :INT:=1;
	
	PRESSURE_REGULATOR_ST4: PRESSURE_REGULATOR;
	PRESSURE_REGULATOR_ST5: PRESSURE_REGULATOR;


END_VAR

// ---- GVLs/IOs_Variables.TcGVL
	{attribute 'Tc2GvlVarNames'}
VAR_GLOBAL


(************************************************************************************************
*
*General
*
***********************************************************************************************)
	PROG_STEPS:PROG_STEPS;
	
	GEN_0B1 				AT%I*:BOOL;		(*Présence AIR*)
	GEN_PRESENCE_POMPE 		AT%I*:BOOL;		(* Une pompe est présente sur la palette à l'entrée du banc*)
	
	GEN_1V1 				AT%Q*:BOOL;		(*Vanne AIR*)
	GEN_CONVOYEUR			AT%Q*:BOOL;		(*Relais convoyeur*)
	
	
	

(************************************************************************************************
*
*Pote 1 - Test haute tension
*
***********************************************************************************************)	
	ST1_1B1 	AT%I*:BOOL;		(*Capteur palette en attente*)
	ST1_1B2 	AT%I*:BOOL;		(*Capteur palette présente*)
	ST1_1B4 	AT%I*:BOOL;		(*Capteur vérin Hydro TOP*)
	ST1_1B5 	AT%I*:BOOL;		(*Capteur vérin Hydro BOTTOM*)
	
	ST1_1V1 	AT%Q*:BOOL;		(*Vérin palette attente*)
	ST1_1V2 	AT%Q*:BOOL;		(*Vérin palette bloquage*)
	ST1_1V3 	AT%Q*:BOOL;		(*Vérin palette stop*)
	ST1_1V4 	AT%Q*:BOOL;		(*Vérin connexion TOP*)
	ST1_1V5		AT%Q*:BOOL;		(*Vérin connexion HT*)
	
	ST1_HT_CTRLIN 	AT%Q*:BOOL;	(*Prise de contrôle par le PLC*)
	ST1_HT_TYPW 	AT%Q*:BOOL;	(*Type de mesure FALSE: Rigidité dielectrique TRUE:Megomètre*)
	ST1_HT_N0		AT%Q*:BOOL;	(*Numéro de programme*)
	ST1_HT_N1 		AT%Q*:BOOL;	(*Numéro de programme*)
	ST1_HT_N2 		AT%Q*:BOOL;	(*Numéro de programme*)
	ST1_HT_MES_DCH 	AT%Q*:BOOL;	(*Passage en mesure / décharge FALSE: Décharge TRUE:Mesure*)
	
	ST1_HT_CTRLOUT 	AT%I*:BOOL;	(*Validation de prise de contrôle par le PLC*)
	ST1_HT_EOT 		AT%I*:BOOL;	(*Fin de test*)
	ST1_HT_PASS 	AT%I*:BOOL;	(*Test BON*)
	ST1_HT_FAIL 	AT%I*:BOOL;	(*Test MAUVAIS*)
	ST1_HT_ERROR 	AT%I*:BOOL;	(*Erreur*)
	
	ST1_HT_OK 		:BOOL;		(*Résultat du test TRUE: Test OK FALSE: Test NOK*)
	
	
	
	
	
(************************************************************************************************
*
*Pote 2 - Aspiration et étanchéité des soupapes
*
***********************************************************************************************)	
	ST2_2B1 	AT%I*:BOOL;		(*Capteur palette en attente*)
	ST2_2B2 	AT%I*:BOOL;		(*Capteur palette présente*)
	ST2_2B4 	AT%I*:BOOL;		(*Capteur vérin Hydro TOP*)
	ST2_2B5 	AT%I*:BOOL;		(*Capteur vérin Hydro BOTTOM*)
	ST2_2B6 	AT%I*:BOOL;		(*Capteur vérin électrique*)
	ST2_2B7 	AT%I*:BOOL;		(*Capteur vérin by-pass*)	
	
	ST2_2P1		AT%I*:PRESSURE_SENSOR; (* Valeurs du capteur aspiration*)
	ST2_VACUUM	:REAL; 					(*Pression aspiration*)
	
	ST2_2V1 	AT%Q*:BOOL;		(*Vérin palette attente*)
	ST2_2V2 	AT%Q*:BOOL;		(*Vérin palette bloquage*)
	ST2_2V3 	AT%Q*:BOOL;		(*Vérin palette stop*)
	ST2_2V4 	AT%Q*:BOOL;		(*Vérin Hydro TOP*)
	ST2_2V5		AT%Q*:BOOL;		(*Vérin hydro BOTTOM*)
	ST2_2V6		AT%Q*:BOOL;		(*Vérin électrique*)
	ST2_2V7		AT%Q*:BOOL;		(*Vérin by-pass*)
	ST2_2V8		AT%Q*:BOOL;		(*Vanne contre pression*)
	
	ST2_POWER	AT%Q*:BOOL;		(*Alimentation électrique pompe*)
	
	
	
(************************************************************************************************
*
*Pote 3 - Etanchéité
*
***********************************************************************************************)	
	ST3_3B1 	AT%I*:BOOL;		(*Capteur palette en attente*)
	ST3_3B2 	AT%I*:BOOL;		(*Capteur palette présente*)
	ST3_3B4 	AT%I*:BOOL;		(*Capteur vérin Hydro TOP*)
	ST3_3B5 	AT%I*:BOOL;		(*Capteur vérin Hydro BOTTOM*)
	ST3_3B7 	AT%I*:BOOL;		(*Capteur vérin by-pass*)	
	
	ST3_3V1 	AT%Q*:BOOL;		(*Vérin palette attente*)
	ST3_3V2 	AT%Q*:BOOL;		(*Vérin palette bloquage*)
	ST3_3V3 	AT%Q*:BOOL;		(*Vérin palette stop*)
	ST3_3V4 	AT%Q*:BOOL;		(*Vérin Hydro TOP*)
	ST3_3V5		AT%Q*:BOOL;		(*Vérin hydro BOTTOM*)
	ST3_3V7		AT%Q*:BOOL;		(*Vérin by-pass*)
	
	ST3_3V10 	AT%Q*:BOOL;		(*Vanne avant la pompe*)
	ST3_3V11 	AT%Q*:BOOL;		(*Vanne après la pompe*)
	ST3_3V12 	AT%Q*:BOOL;		(*Vanne de blocage d'air pour le DELTA*)
	
	ST3_3P1 	AT%I*:INT;		(*Capteur de pression différentiel*)
	ST3_3P2		AT%I*:INT;		(*Capteur de pression absolue pour détecter les grandes fuites*)
	ST3_PRESSION	:REAL;		(*Capteur de pression différentiel - Valeur réel en mBar*)
	ST3_PRESSION_ABS:REAL;		(*Capteur de pression absolue - valeur réel en mBar*)
	
	ST3_DELTA_P	:REAL;			(*Mesure de la chutte de pression en mbar*)
	ST3_DELTA_P_ABS: REAL;		(*Mesure grossière de la chute de pression en mbar*)
	ST3_PRESSION_FIN_ABS: REAL; 

(************************************************************************************************
*
*Pote 4 et 5  - Débits - Variables pour HMI
*
**********************************************************************************************)	
	ST45_QMAX		:REAL;			(*Débit max calculé*)
	ST45_Q			:REAL;			(*Débit travail calculé*)
	ST45_PRESSURE	:REAL; 			(*Pression fitré*)
	ST45_VACUUM		:REAL; 			(*Pression aspiration*)
	ST45_POIDS		:REAL;			(*Poids sur la balance*)
	
	ST45_COURANT	:REAL;			(*Courant*)
	
(************************************************************************************************
*
*Pote 4 - Débit (petit)
*
**********************************************************************************************)	
	ST4_4B1 	AT%I*:BOOL;		(*Capteur palette en attente*)
	ST4_4B2 	AT%I*:BOOL;		(*Capteur palette présente*)
	ST4_4B4 	AT%I*:BOOL;		(*Capteur vérin Hydro TOP*)
	ST4_4B5 	AT%I*:BOOL;		(*Capteur vérin Hydro BOTTOM*)
	ST4_4B6 	AT%I*:BOOL;		(*Capteur vérin électrique*)
	ST4_4B7 	AT%I*:BOOL;		(*Capteur vérin by-pass*)	
	
	ST4_4P1			AT%I*:PRESSURE_SENSOR; 	(*Valeurs du capteur*)
	ST4_VACUUM		:REAL; 					(*Pression aspiration*)
	
	ST4_4P2					AT%I*:PRESSURE_SENSOR; 	(*Valeurs du capteur*)
	ST4_PRESSURE			:REAL; 					(*Pression*)
	ST4_PRESSURE_FILTERED	:REAL; 					(*Pression fitré*)
	
	ST4_POIDS 			AT%I*:REAL;		(*Poids balance*)	
	ST4_QMAX	:REAL;			(*Débit max calculé*)
	ST4_Q		:REAL;			(*Débit travail calculé*)
	
	ST4_COURANT	:REAL;			(*Courant*)
	
	ST4_DIGMESA	AT%I*:BOOL;		(*Digmesa*)
	
	ST4_4V1 	AT%Q*:BOOL;		(*Vérin palette attente*)
	ST4_4V2 	AT%Q*:BOOL;		(*Vérin palette bloquage*)
	ST4_4V3 	AT%Q*:BOOL;		(*Vérin palette stop*)
	ST4_4V4 	AT%Q*:BOOL;		(*Vérin Hydro TOP*)
	ST4_4V5		AT%Q*:BOOL;		(*Vérin hydro BOTTOM*)
	ST4_4V6		AT%Q*:BOOL;		(*Vérin électrique*)
	ST4_4V7		AT%Q*:BOOL;		(*Vérin by-pass*)
	
	ST4_4V10	AT%Q*:BOOL;		(*Vanne avant la pompe*)
	ST4_4V12	AT%Q*:BOOL;		(*Vanne après la vanne pilotée*)
	ST4_4V13	AT%Q*:BOOL;		(*Vanne max flow*)

	ST4_POWER	AT%Q*:BOOL;		(*Alimentation électrique pompe*)
	ST4_VIDANGE	AT%Q*:BOOL;		(*Vidange balance*)

(************************************************************************************************
*
*Pote 5 - Débit (grand)
*
***********************************************************************************************)	
	ST5_5B1 	AT%I*:BOOL;		(*Capteur palette en attente*)
	ST5_5B2 	AT%I*:BOOL;		(*Capteur palette présente*)
	ST5_5B4 	AT%I*:BOOL;		(*Capteur vérin Hydro TOP*)
	ST5_5B5 	AT%I*:BOOL;		(*Capteur vérin Hydro BOTTOM*)
	ST5_5B6 	AT%I*:BOOL;		(*Capteur vérin électrique*)	
	
	ST5_5P1			AT%I*:PRESSURE_SENSOR; 	(*Valeurs du capteur*)
	ST5_VACUUM		:REAL; 					(*Pression aspiration*)
	
	ST5_5P2			AT%I*:PRESSURE_SENSOR; 	(*Valeurs du capteur*)
	ST5_PRESSURE	:REAL; 					(*Pression aspiration*)
	ST5_PRESSURE_FILTERED	:REAL; 					(*Pression fitré*)
	
	ST5_POIDS 			AT%I*:REAL;		(*Poids balance*)	
	ST5_QMAX	:REAL;			(*Débit max calculé*)
	ST5_Q		:REAL;			(*Débit travail calculé*)
	
	ST5_COURANT	:REAL;			(*Courant*)
	
	ST5_5V1 	AT%Q*:BOOL;		(*Vérin palette attente*)
	ST5_5V2 	AT%Q*:BOOL;		(*Vérin palette bloquage*)
	ST5_5V3 	AT%Q*:BOOL;		(*Vérin palette stop*)
	ST5_5V4 	AT%Q*:BOOL;		(*Vérin Hydro TOP*)
	ST5_5V5		AT%Q*:BOOL;		(*Vérin hydro BOTTOM*)
	ST5_5V6		AT%Q*:BOOL;		(*Vérin électrique*)
	
	ST5_5V10	AT%Q*:BOOL;		(*Vanne avant la pompe*)
	ST5_5V12	AT%Q*:BOOL;		(*Vanne après la vanne pilotée*)
	ST5_5V13	AT%Q*:BOOL;		(*Vanne max flow*)
	
	ST5_5V14	AT%Q*:BOOL;		(*Vanne vidange vers égouts ou réservoir*)
	ST5_5V15	AT%Q*:BOOL;		(*Vanne avant la pompe*)
	ST5_5V16	AT%Q*:BOOL;		(*Vanne provenance eau du réservoir ou du déminéralisateur*)
	
	ST5_POWER	AT%Q*:BOOL;		(*Alimentation électrique pompe*)
	ST5_VIDANGE	AT%Q*:BOOL;		(*Vidange balance*)
	
	ST5_Niveau_Reservoir 	AT%I*:INT; (*Niveau réservoir - valeur du capteur*)
	
	ST5_MODE_VIDANGE		:INT:=1;(*Mode de vidange 1-Mode normal 2-Vidange du réseroir 3-Remplissage depuis le banc déminéralisateur*)
	ST5_NIVEAU_EAU			:INT;	(*Niveau du réservoir 0-100%*)
	

(************************************************************************************************
*
*Pote 6 - Pression max
*
***********************************************************************************************)	
	ST6_6B1 	AT%I*:BOOL;		(*Capteur palette en attente*)
	ST6_6B2 	AT%I*:BOOL;		(*Capteur palette présente*)
	ST6_6B4 	AT%I*:BOOL;		(*Capteur vérin Hydro TOP*)
	ST6_6B5 	AT%I*:BOOL;		(*Capteur vérin Hydro BOTTOM*)
	ST6_6B6 	AT%I*:BOOL;		(*Capteur vérin électrique*)
	ST6_6B7 	AT%I*:BOOL;		(*Capteur vérin by-pass*)	
	
	ST6_6P1			AT%I*:PRESSURE_SENSOR; 	(*Valeurs du capteur*)
	ST6_PRESSURE	:REAL; 					(*Pression*)
	
	ST6_6V1 	AT%Q*:BOOL;		(*Vérin palette attente*)
	ST6_6V2 	AT%Q*:BOOL;		(*Vérin palette bloquage*)
	ST6_6V3 	AT%Q*:BOOL;		(*Vérin palette stop*)
	ST6_6V4 	AT%Q*:BOOL;		(*Vérin Hydro TOP*)
	ST6_6V5		AT%Q*:BOOL;		(*Vérin hydro BOTTOM*)
	ST6_6V6		AT%Q*:BOOL;		(*Vérin électrique*)
	ST6_6V7		AT%Q*:BOOL;		(*Vérin by-pass*)
	
	ST6_6V10	AT%Q*:BOOL;		(*Vanne avant la pompe*)
	ST6_6V11	AT%Q*:BOOL;		(*Vanne après la pompe*)
	
	ST6_POWER	AT%Q*:BOOL;		(*Alimentation électrique pompe*)
	
(************************************************************************************************
*
*Pote 7 - Séchage
*
***********************************************************************************************)	
	ST7_7B1 	AT%I*:BOOL;		(*Capteur palette en attente*)
	ST7_7B2 	AT%I*:BOOL;		(*Capteur palette présente*)
	ST7_7B4 	AT%I*:BOOL;		(*Capteur vérin Hydro TOP*)
	ST7_7B5 	AT%I*:BOOL;		(*Capteur vérin Hydro BOTTOM*)
	ST7_7B6 	AT%I*:BOOL;		(*Capteur vérin électrique*)
	ST7_7B7 	AT%I*:BOOL;		(*Capteur vérin by-pass*)	
	
	ST7_RESERVE	AT%Q*:BOOL;		(*Vanne de réserve*)
	ST7_7V1 	AT%Q*:BOOL;		(*Vérin palette attente*)
	ST7_7V2 	AT%Q*:BOOL;		(*Vérin palette bloquage*)
	ST7_7V3 	AT%Q*:BOOL;		(*Vérin palette stop*)
	ST7_7V4 	AT%Q*:BOOL;		(*Vérin Hydro TOP*)
	ST7_7V5		AT%Q*:BOOL;		(*Vérin hydro BOTTOM*)
	ST7_7V6		AT%Q*:BOOL;		(*Vérin électrique*)
	ST7_7V7		AT%Q*:BOOL;		(*Vérin by-pass*)
	
	ST7_7V10	AT%Q*:BOOL;		(*Vanne avant la pompe*)
	
	ST7_POWER	AT%Q*:BOOL;		(*Alimentation électrique pompe*)

(************************************************************************************************
*
*Pote 8  - Etiquettage
*
***********************************************************************************************)	
	ST8_8B1 	AT%I*:BOOL;		(*Capteur palette en attente*)
	ST8_8B2 	AT%I*:BOOL;		(*Capteur palette présente*)
	
	ST8_8V1 	AT%Q*:BOOL;		(*Vérin palette attente*)
	ST8_8V2 	AT%Q*:BOOL;		(*Vérin palette bloquage*)
	ST8_8V3 	AT%Q*:BOOL;		(*Vérin palette stop*)
	ST8_8V4 	AT%Q*:BOOL;		(*Reserve*)
	
	ST8_PRET_A_IMPRIMER :BOOL;	(*Pompe prête pour l'impression de l'étiquette*)
	ST8_IMPRESSION_OK	:BOOL;	(*L'impression de l'étiquette a été effectuée*)
	
(************************************************************************************************
*
*Pote 9  - Déchagement
*
***********************************************************************************************)	
	ST9_9B1 	AT%I*:BOOL;		(*Capteur palette en attente*)
	ST9_9B2 	AT%I*:BOOL;		(*Capteur palette présente*)
	ST9_9B4 	AT%I*:BOOL;		(*Capteur rodless guide DECHARGEMENT*)
	ST9_9B41 	AT%I*:BOOL;		(*Capteur rodless guide PALETTE*)
	ST9_9B5 	AT%I*:BOOL;		(*Capteur slide table HAUT*)
	ST9_9B51 	AT%I*:BOOL;		(*Capteur slide table BAS*)
	ST9_9B6 	AT%I*:BOOL;		(*Capteur gripper OPENED*)	
	ST9_9B61 	AT%I*:BOOL;		(*Capteur gripper CLOSED*)
	ST9_9B7 	AT%I*:BOOL;		(*Capteur vérin libération connecteurs électriques*)
	
	ST9_9V1 	AT%Q*:BOOL;		(*Vérin palette attente*)
	ST9_9V2 	AT%Q*:BOOL;		(*Vérin palette bloquage*)
	ST9_9V3 	AT%Q*:BOOL;		(*Vérin palette stop*)
	ST9_9V4A 	AT%Q*:BOOL;		(*Vérin vers palette*)
	ST9_9V4B 	AT%Q*:BOOL;		(*Vérin vers palette*)
	ST9_9V5A 	AT%Q*:BOOL;		(*Vérin vers déchargement*)
	ST9_9V5B 	AT%Q*:BOOL;		(*Vérin vers déchargement*)
	ST9_9V6 	AT%Q*:BOOL;		(*Vérin descend*)
	ST9_9V7 	AT%Q*:BOOL;		(*Vérin monte*)
	
	ST9_DECHARGE 	AT%Q*:BOOL;		(*TRUE - décharge / FALSE - pas décharge*)
	
	
(************************************************************************************************
*
*Convoyeur
*
***********************************************************************************************)	
	ST10_10B1 	AT%I*:BOOL;		(*Opérateur 1 - Palette présente*)
	ST10_10B2 	AT%I*:BOOL;		(*Opérateur 2 - Palette présente*)
	ST10_OPERATEUR1_START 	AT%I*:BOOL; (* Pédale pour l'opérateur 1*)
	ST10_OPERATEUR2_START	AT%I*:BOOL; (* Pédale pour l'opérateur 2*)
	
	ST10_10V1 	AT%Q*:BOOL;		(*Opérateur 1 - Vérin carrier stop*)
	ST10_10V2 	AT%Q*:BOOL;		(*Opérateur 2 - Vérin carrier stop*)
	


(************************************************************************************************
*
*Current measurement
*
***********************************************************************************************)
	ST4_Multimeter_mode	AT%Q*:SINT := 3;
	ST5_Multimeter_mode	AT%Q*:SINT := 3;
(*
0 0x00 DC voltage
1 0x01 AC voltage
2 0x02 DC current
3 0x03 AC current
*)
	ST4_Multimeter_range AT%Q* :SINT := 1;
	ST5_Multimeter_range AT%Q* :SINT := 1;
(*
255 0xFF 300 mV / 100 mA
0 0x00  3 V / 1 A 
1 0x01 30 V / 10 A 
2 0x02 300 V (voltage only)  
*)
	ST4_Multimeter_value AT%I*:DINT;
	ST5_Multimeter_value AT%I*:DINT;


END_VAR

// ---- GVLs/PID_parameters.TcGVL
VAR_GLOBAL
	(* q is the gain scheduling parameter, here the operating pressure *)
	ST4_PID_LowPressure		:GAIN_SCHEDULED_PID	:= (q:=0.8,Kp:=3,Ki:=1.4,Kd:=15); 
	ST4_PID_HighPressure	:GAIN_SCHEDULED_PID	:= (q:=8,Kp:=0.5,Ki:=1.6,Kd:=30); 
	ST4_PID_MiddlePressure	:GAIN_SCHEDULED_PID	:= (q:=4,Kp:=1.35,Ki:=5.25,Kd:=35);
	
	ST5_PID_MiddlePressure	:GAIN_SCHEDULED_PID	:= (q:=1.5,Kp:=0.8,Ki:=1.7,Kd:=2); 
	ST5_PID_LowPressure		:GAIN_SCHEDULED_PID	:= (q:=0.7,Kp:=2.2,Ki:=1.4,Kd:=2); 
	
END_VAR

(***** backup *****
	ST4_PID_LowPressure		:GAIN_SCHEDULED_PID	:= (q:=0.8,Kp:=3,Ki:=1.4,Kd:=15); 
	ST4_PID_HighPressure	:GAIN_SCHEDULED_PID	:= (q:=8,Kp:=0.5,Ki:=1.6,Kd:=30); 
	ST4_PID_MiddlePressure	:GAIN_SCHEDULED_PID	:= (q:=4,Kp:=1.35,Ki:=5.25,Kd:=35);
*)

// ---- POUs/MAIN.TcPOU
PROGRAM MAIN
VAR
	ST4_VIDANGE_BALANCE: VIDANGE_BALANCE_ST4;
	ST5_VIDANGE_BALANCE: VIDANGE_BALANCE_ST5;
END_VAR

(*Appel les différents modules généraux*)
SAFETY();
GEMMA();
CONVEYOR();
AIS();
ST45_TO_HMI();

ST4_MOTOR();
ST5_MOTOR();

(*Appel les différents modules pour les stations*)
ST1_HT();
ST2_ASPIRATION();
ST3_ETANCHEITE();
ST4_DEBIT_PETIT();
ST5_GRAND_PETIT();
ST6_PMAX();
ST7_SECHAGE();
ST8_IMPRESSION();
ST9_DECHARGEMENT();

(*Gestion de la vidange de la balance ST4*)
ST4_VIDANGE_BALANCE(
PROG_STEP:= PROG_STEPS.ST4,
POIDS:= ST4_POIDS, 
POIDS_LIMIT:= BALANCE_POIDS_LIMITE, 
POMPE=> ST4_VIDANGE);

(*Gestion de la vidange de la balance ST5*)
ST5_VIDANGE_BALANCE(
MODE:= ST5_MODE_VIDANGE, 
PROG_STEP:= PROG_STEPS.ST5,
POIDS:= ST5_POIDS, 
POIDS_LIMIT:= BALANCE_POIDS_LIMITE, 
POMPE=> ST5_VIDANGE);

END_PROGRAM

// ---- POUs/EAU/VIDANGE_BALANCE_ST4.TcPOU
FUNCTION_BLOCK VIDANGE_BALANCE_ST4
VAR_INPUT
	POIDS: REAL;
	POIDS_LIMIT: REAL;
	PROG_STEP: INT;
END_VAR
VAR_OUTPUT
	POMPE: BOOL;
END_VAR
VAR
	POMPE_START: BOOL;
	POMPE_STOP: BOOL;

END_VAR

IF ((POIDS+200) > POIDS_LIMIT) AND (GEMMA.STEP='F1' OR GEMMA.STEP='A1')  AND (PROG_STEP<100 OR PROG_STEP>=300) THEN (*Hystérésis de 200g*)

	POMPE	:= TRUE; 

ELSIF (POIDS < POIDS_LIMIT) AND (GEMMA.STEP='F1' OR GEMMA.STEP='A1') AND (PROG_STEP<100 OR PROG_STEP>=300) THEN

	POMPE 	:= FALSE;
	
ELSE
	
	POMPE 	:= FALSE;

END_IF;

END_FUNCTION_BLOCK

// ---- POUs/GEMMA.TcPOU
PROGRAM GEMMA
VAR
	STEP_A6: INT := 0;
	DELAY_EJECTION_CARRIERS: TON;
	DELAY_STARTING_AIR: TON;
	EJECT_CARRIERS: BOOL;
	F2_END: BOOL;
	STEP: STRING(20);
	START_AIR: BOOL;
END_VAR

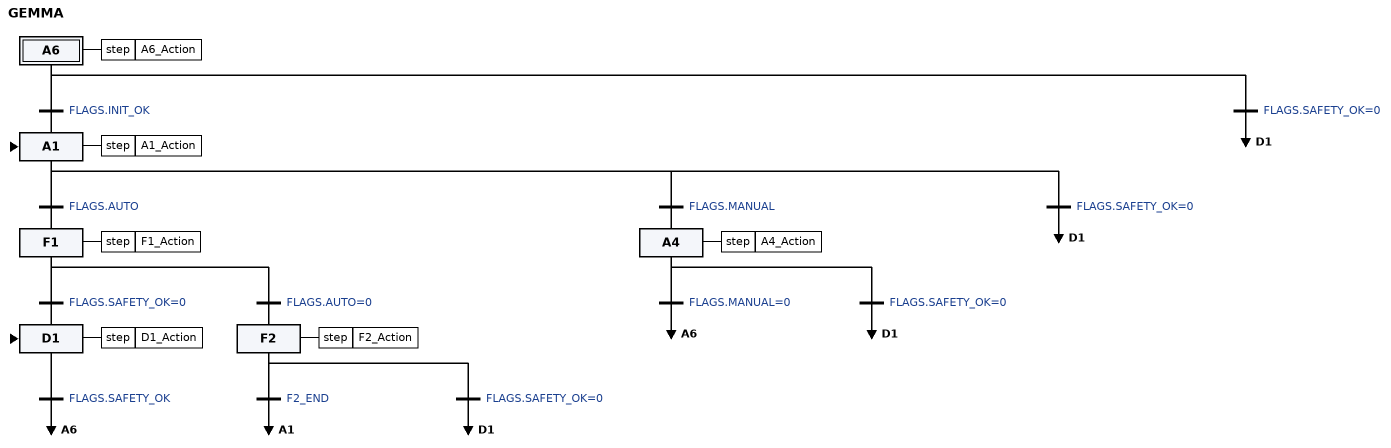
INITIAL_STEP A6_:  // name as stored: A6 
    A6_Action(N);  // step action
END_STEP
TRANSITION FROM A6_ TO A1
    := FLAGS.INIT_OK;
END_TRANSITION
TRANSITION FROM A6_ TO D1
    := FLAGS.SAFETY_OK=0;
END_TRANSITION
STEP A1:
    A1_Action(N);  // step action
END_STEP
TRANSITION FROM A1 TO F1
    := FLAGS.AUTO;
END_TRANSITION
TRANSITION FROM A1 TO A4
    := FLAGS.MANUAL;
END_TRANSITION
STEP A4:
    A4_Action(N);  // step action
END_STEP
TRANSITION FROM A4 TO A6
    := FLAGS.MANUAL=0;
END_TRANSITION
TRANSITION FROM A4 TO D1
    := FLAGS.SAFETY_OK=0;
END_TRANSITION
TRANSITION FROM A1 TO D1
    := FLAGS.SAFETY_OK=0;
END_TRANSITION
STEP F1:
    F1_Action(N);  // step action
END_STEP
TRANSITION FROM F1 TO D1
    := FLAGS.SAFETY_OK=0;
END_TRANSITION
TRANSITION FROM F1 TO F2
    := FLAGS.AUTO=0;
END_TRANSITION
STEP F2:
    F2_Action(N);  // step action
END_STEP
TRANSITION FROM F2 TO A1
    := F2_END;
END_TRANSITION
TRANSITION FROM F2 TO D1
    := FLAGS.SAFETY_OK=0;
END_TRANSITION
STEP D1:
    D1_Action(N);  // step action
END_STEP
TRANSITION FROM D1 TO A6
    := FLAGS.SAFETY_OK;
END_TRANSITION

ACTION F1_Action:
(*********************************************************
*
* F1
*
************************************************************)

STEP := 'F1';
END_ACTION

ACTION A6_Action:
(**************************************************************
*
*
* Initialisation
*
*
***************************************************************)
STEP:='A6';



CASE STEP_A6 OF

0: (*Init*)
	STEP_A6:=STEP_A6+1;

1: (*Initialise valves and variables*)

	GEN_1V1 				:=FALSE;	(*Vanne AIR*)
	GEN_CONVOYEUR			:=FALSE;	(*Relais convoyeur*)	
	
	ST1_1V1 	:=FALSE;		(*Vérin palette attente*)
	ST1_1V2 	:=FALSE;		(*Vérin palette bloquage*)
	ST1_1V3 	:=FALSE;		(*Vérin palette stop*)
	ST1_1V4 	:=FALSE;		(*Vérin connexion TOP*)
	ST1_1V5		:=FALSE;		(*Vérin connexion HT*)

	ST2_2V1 	:=FALSE;		(*Vérin palette attente*)
	ST2_2V2 	:=FALSE;		(*Vérin palette bloquage*)
	ST2_2V3 	:=FALSE;		(*Vérin palette stop*)
	ST2_2V4 	:=FALSE;		(*Vérin Hydro TOP*)
	ST2_2V5		:=FALSE;		(*Vérin hydro BOTTOM*)
	ST2_2V6		:=FALSE;		(*Vérin électrique*)
	ST2_2V7		:=FALSE;		(*Vérin by-pass*)
	
	ST2_POWER	:=FALSE;		(*Alimentation électrique pompe*)
	
	ST3_3V1 	:=FALSE;		(*Vérin palette attente*)
	ST3_3V2 	:=FALSE;		(*Vérin palette bloquage*)
	ST3_3V3 	:=FALSE;		(*Vérin palette stop*)
	ST3_3V4 	:=FALSE;		(*Vérin Hydro TOP*)
	ST3_3V5		:=FALSE;		(*Vérin hydro BOTTOM*)
	ST3_3V7		:=FALSE;		(*Vérin by-pass*)
	
	ST3_3V10 	:=FALSE;		(*Vanne avant la pompe*)
	ST3_3V11 	:=FALSE;		(*Vanne après la pompe*)
	ST3_3V12 	:=FALSE;		(*Vanne de blocage d'air pour le DELTA*)
	
	ST4_4V1 	:=FALSE;		(*Vérin palette attente*)
	ST4_4V2 	:=FALSE;		(*Vérin palette bloquage*)
	ST4_4V3 	:=FALSE;		(*Vérin palette stop*)
	ST4_4V4 	:=FALSE;		(*Vérin Hydro TOP*)
	ST4_4V5		:=FALSE;		(*Vérin hydro BOTTOM*)
	ST4_4V6		:=FALSE;		(*Vérin électrique*)
	ST4_4V7		:=FALSE;		(*Vérin by-pass*)
	
	ST4_4V10	:=FALSE;		(*Vanne avant la pompe*)
	ST4_4V12	:=FALSE;		(*Vanne après la vanne pilotée*)
	ST4_4V13	:=FALSE;		(*Vanne max flow*)

	ST4_POWER	:=FALSE;		(*Alimentation électrique pompe*)
	ST4_VIDANGE	:=FALSE;		(*Vidange balance*)
	
	ST5_5V1 	:=FALSE;		(*Vérin palette attente*)
	ST5_5V2 	:=FALSE;		(*Vérin palette bloquage*)
	ST5_5V3 	:=FALSE;		(*Vérin palette stop*)
	ST5_5V4 	:=FALSE;		(*Vérin Hydro TOP*)
	ST5_5V5		:=FALSE;		(*Vérin hydro BOTTOM*)
	ST5_5V6		:=FALSE;		(*Vérin électrique*)
	
	ST5_5V10	:=FALSE;		(*Vanne avant la pompe*)
	ST5_5V12	:=FALSE;		(*Vanne après la vanne pilotée*)
	ST5_5V13	:=FALSE;		(*Vanne max flow*)
	
	ST5_5V14	:=FALSE;		(*Vanne vidange vers égouts ou réservoir*)
	ST5_5V15	:=FALSE;			(*Vanne avant la pompe*)
	ST5_5V16	:=FALSE;		(*Vanne provenance eau du réservoir ou du déminéralisateur*)
	
	ST5_POWER	:=FALSE;		(*Alimentation électrique pompe*)
	ST5_VIDANGE	:=FALSE;		(*Vidange balance*)
	
	ST6_6V1 	:=FALSE;		(*Vérin palette attente*)
	ST6_6V2 	:=FALSE;		(*Vérin palette bloquage*)
	ST6_6V3 	:=FALSE;		(*Vérin palette stop*)
	ST6_6V4 	:=FALSE;		(*Vérin Hydro TOP*)
	ST6_6V5		:=FALSE;		(*Vérin hydro BOTTOM*)
	ST6_6V6		:=FALSE;		(*Vérin électrique*)
	ST6_6V7		:=FALSE;		(*Vérin by-pass*)
	
	ST6_6V10	:=FALSE;		(*Vanne avant la pompe*)
	ST6_6V11	:=FALSE;		(*Vanne après la pompe*)
	
	ST6_POWER	:=FALSE;		(*Alimentation électrique pompe*)
	
	ST7_7V1 	:=FALSE;		(*Vérin palette attente*)
	ST7_7V2 	:=FALSE;		(*Vérin palette bloquage*)
	ST7_7V3 	:=FALSE;		(*Vérin palette stop*)
	ST7_7V4 	:=FALSE;		(*Vérin Hydro TOP*)
	ST7_7V5		:=FALSE;		(*Vérin hydro BOTTOM*)
	ST7_7V6		:=FALSE;		(*Vérin électrique*)
	ST7_7V7		:=FALSE;		(*Vérin by-pass*)
	
	ST7_7V10	:=FALSE;		(*Vanne avant la pompe*)
	
	ST7_POWER	:=FALSE;		(*Alimentation électrique pompe*)
	
	ST8_8V1 	:=FALSE;		(*Vérin palette attente*)
	ST8_8V2 	:=FALSE;		(*Vérin palette bloquage*)
	ST8_8V3 	:=FALSE;		(*Vérin palette stop*)
	ST8_8V4 	:=FALSE;		(*Reserve*)
	
	ST9_9V1 	:=FALSE;		(*Vérin palette attente*)
	ST9_9V2 	:=FALSE;		(*Vérin palette bloquage*)
	ST9_9V3 	:=FALSE;		(*Vérin palette stop*)
	ST9_9V4A 	:=TRUE;			(*Vérin rodless guide*)
	ST9_9V4B 	:=FALSE;		(*Vérin rodless guide*)
	ST9_9V5A 	:=FALSE;		(*Vérin slide table*)
	ST9_9V5B 	:=TRUE;			(*Vérin slide table*)
	ST9_9V6 	:=TRUE;			(*Vérin gripper*)
	ST9_9V7 	:=FALSE;		(*Vérin liberateur electrique*)
	
	ST10_10V1 	:=TRUE;		(*Opérateur 1 - Vérin carrier stop*)
	ST10_10V2 	:=TRUE;		(*Opérateur 2 - Vérin carrier stop*)
	
	FLAGS.MOTOR_ST4_POSITION := MOTOR_ST4_INITIAL_POS;
	FLAGS.MOTOR_ST5_POSITION := MOTOR_ST5_INITIAL_POS;


	STEP_A6:=STEP_A6+1;

2: (*Start AIR*)

	GEN_1V1 := TRUE;
	START_AIR := TRUE;
	STEP_A6:=STEP_A6+1;

3: (*Wait AIR then start convoyer and wait ejection of carriers*)
	
	IF DELAY_STARTING_AIR.Q THEN
		GEN_CONVOYEUR := TRUE;
		START_AIR := FALSE;
		EJECT_CARRIERS:=TRUE;
		STEP_A6:=STEP_A6+1;
	END_IF;

4: (* Wait carriers ejection *)

	IF DELAY_EJECTION_CARRIERS.Q AND GEN_0B1 THEN
		EJECT_CARRIERS:=FALSE;
		STEP_A6:=STEP_A6+1;
	END_IF;
5: (*End of init *)

	FLAGS.INIT_OK:=TRUE;


ELSE
    ;
END_CASE;

(* FBs *)
DELAY_EJECTION_CARRIERS(IN:=EJECT_CARRIERS , PT:=DELAY_EJECT_CARRIERS);
DELAY_STARTING_AIR(IN:=START_AIR , PT:=DELAY_START_AIR);
END_ACTION

ACTION A1_Action:
(***************************************************************************
*
* A1
*
****************************************************************************)
STEP := 'A1';

(*Réglage pression**********************************************)
PRESSURE_REGULATOR_ST4(
GEMMA				:= GEMMA.STEP,
COURANT				:= ST4_COURANT, 
PRESSION_CONSIGNE	:= PUMP_PARAMS.ST45_PRESSION_CONSIGNE, 
PRESSION_MESURE		:= ST4_PRESSURE_FILTERED,
MOTOR_POSITION_MAX	:= MOTOR_ST4_POSITION_MAX,
MOTOR_INITIAL_POSITION := MOTOR_ST4_INITIAL_POS,
MOTOR_POSITION		=> FLAGS.MOTOR_ST4_POSITION
);
END_ACTION

ACTION A4_Action:
STEP:= 'A4';
END_ACTION

ACTION D1_Action:
(*****************************************************************
*
* NOT AUS state
*
******************************************************************)

	STEP := 'D1';
	
	STEP_A6:=0;
	F2_END:=FALSE;

	FLAGS.INIT_OK			:=FALSE;
	FLAGS.MOTOR_ST4_INIT_OK	:=FALSE;
	FLAGS.AUTO				:=FALSE;
	FLAGS.MANUAL			:=FALSE;

	GEN_1V1 				:=FALSE;	(*Vanne AIR*)
	GEN_CONVOYEUR			:=FALSE;	(*Relais convoyeur*)	
	
	ST1_1V1 	:=FALSE;		(*Vérin palette attente*)
	ST1_1V2 	:=FALSE;		(*Vérin palette bloquage*)
	ST1_1V3 	:=FALSE;		(*Vérin palette stop*)
	ST1_1V4 	:=FALSE;		(*Vérin connexion TOP*)
	ST1_1V5		:=FALSE;		(*Vérin connexion HT*)

	ST2_2V1 	:=FALSE;		(*Vérin palette attente*)
	ST2_2V2 	:=FALSE;		(*Vérin palette bloquage*)
	ST2_2V3 	:=FALSE;		(*Vérin palette stop*)
	ST2_2V4 	:=FALSE;		(*Vérin Hydro TOP*)
	ST2_2V5		:=FALSE;		(*Vérin hydro BOTTOM*)
	ST2_2V6		:=FALSE;		(*Vérin électrique*)
	ST2_2V7		:=FALSE;		(*Vérin by-pass*)
	
	ST2_POWER	:=FALSE;		(*Alimentation électrique pompe*)
	
	ST3_3V1 	:=FALSE;		(*Vérin palette attente*)
	ST3_3V2 	:=FALSE;		(*Vérin palette bloquage*)
	ST3_3V3 	:=FALSE;		(*Vérin palette stop*)
	ST3_3V4 	:=FALSE;		(*Vérin Hydro TOP*)
	ST3_3V5		:=FALSE;		(*Vérin hydro BOTTOM*)
	ST3_3V7		:=FALSE;		(*Vérin by-pass*)
	
	ST3_3V10 	:=FALSE;		(*Vanne avant la pompe*)
	ST3_3V11 	:=FALSE;		(*Vanne après la pompe*)
	ST3_3V12 	:=FALSE;		(*Vanne de blocage d'air pour le DELTA*)
	
	ST4_4V1 	:=FALSE;		(*Vérin palette attente*)
	ST4_4V2 	:=FALSE;		(*Vérin palette bloquage*)
	ST4_4V3 	:=FALSE;		(*Vérin palette stop*)
	ST4_4V4 	:=FALSE;		(*Vérin Hydro TOP*)
	ST4_4V5		:=FALSE;		(*Vérin hydro BOTTOM*)
	ST4_4V6		:=FALSE;		(*Vérin électrique*)
	ST4_4V7		:=FALSE;		(*Vérin by-pass*)
	
	ST4_4V10	:=FALSE;		(*Vanne avant la pompe*)
	ST4_4V12	:=FALSE;		(*Vanne après la vanne pilotée*)
	ST4_4V13	:=FALSE;		(*Vanne max flow*)

	ST4_POWER	:=FALSE;		(*Alimentation électrique pompe*)
	ST4_VIDANGE	:=FALSE;		(*Vidange balance*)
	
	ST5_5V1 	:=FALSE;		(*Vérin palette attente*)
	ST5_5V2 	:=FALSE;		(*Vérin palette bloquage*)
	ST5_5V3 	:=FALSE;		(*Vérin palette stop*)
	ST5_5V4 	:=TRUE;			(*Vérin Hydro TOP*)
	ST5_5V5		:=FALSE;		(*Vérin hydro BOTTOM*)
	ST5_5V6		:=FALSE;		(*Vérin électrique*)
	
	ST5_5V10	:=FALSE;		(*Vanne avant la pompe*)
	ST5_5V12	:=FALSE;		(*Vanne après la vanne pilotée*)
	ST5_5V13	:=FALSE;		(*Vanne max flow*)
	
	ST5_5V14	:=FALSE;		(*Vanne vidange vers égouts ou réservoir*)
	ST5_5V15	:=FALSE;			(*Vanne avant la pompe*)
	ST5_5V16	:=FALSE;		(*Vanne provenance eau du réservoir ou du déminéralisateur*)
	
	ST5_POWER	:=FALSE;		(*Alimentation électrique pompe*)
	ST5_VIDANGE	:=FALSE;		(*Vidange balance*)
	
	ST6_6V1 	:=FALSE;		(*Vérin palette attente*)
	ST6_6V2 	:=FALSE;		(*Vérin palette bloquage*)
	ST6_6V3 	:=FALSE;		(*Vérin palette stop*)
	ST6_6V4 	:=FALSE;		(*Vérin Hydro TOP*)
	ST6_6V5		:=FALSE;		(*Vérin hydro BOTTOM*)
	ST6_6V6		:=FALSE;		(*Vérin électrique*)
	ST6_6V7		:=FALSE;		(*Vérin by-pass*)
	
	ST6_6V10	:=FALSE;		(*Vanne avant la pompe*)
	ST6_6V11	:=FALSE;		(*Vanne après la pompe*)
	
	ST6_POWER	:=FALSE;		(*Alimentation électrique pompe*)
	
	ST7_7V1 	:=FALSE;		(*Vérin palette attente*)
	ST7_7V2 	:=FALSE;		(*Vérin palette bloquage*)
	ST7_7V3 	:=FALSE;		(*Vérin palette stop*)
	ST7_7V4 	:=FALSE;		(*Vérin Hydro TOP*)
	ST7_7V5		:=FALSE;		(*Vérin hydro BOTTOM*)
	ST7_7V6		:=FALSE;		(*Vérin électrique*)
	ST7_7V7		:=FALSE;		(*Vérin by-pass*)
	
	ST7_7V10	:=FALSE;		(*Vanne avant la pompe*)
	
	ST7_POWER	:=FALSE;		(*Alimentation électrique pompe*)
	
	ST8_8V1 	:=FALSE;		(*Vérin palette attente*)
	ST8_8V2 	:=FALSE;		(*Vérin palette bloquage*)
	ST8_8V3 	:=FALSE;		(*Vérin palette stop*)
	ST8_8V4 	:=FALSE;		(*Reserve*)
	
	ST9_9V1 	:=FALSE;		(*Vérin palette attente*)
	ST9_9V2 	:=FALSE;		(*Vérin palette bloquage*)
	ST9_9V3 	:=FALSE;		(*Vérin palette stop*)
	ST9_9V4A 	:=TRUE;			(*Vérin rodless guide*)
	ST9_9V4B 	:=FALSE;		(*Vérin rodless guide*)
	ST9_9V5A 	:=FALSE;		(*Vérin slide table*)
	ST9_9V5B 	:=TRUE;			(*Vérin slide table*)
	ST9_9V6 	:=TRUE;			(*Vérin gripper*)
	ST9_9V7 	:=FALSE;		(*Vérin liberateur electrique*)
	
	ST10_10V1 	:=TRUE;		(*Opérateur 1 - Vérin carrier stop*)
	ST10_10V2 	:=TRUE;		(*Opérateur 2 - Vérin carrier stop*)
END_ACTION

ACTION F2_Action:
STEP := 'F2';
END_ACTION

END_PROGRAM

// ---- POUs/EAU/VIDANGE_BALANCE_ST5.TcPOU
FUNCTION_BLOCK VIDANGE_BALANCE_ST5
VAR_INPUT
	POIDS: REAL;
	POIDS_LIMIT: REAL;
	PROG_STEP: INT;
	MODE:INT;
END_VAR
VAR_OUTPUT
	POMPE: BOOL;
END_VAR
VAR
	POMPE_START: BOOL;
	POMPE_STOP: BOOL;

	TAMPO_VIDANGE_TON: TON;
	START_TAMPO_VIDANGE: BOOL;
END_VAR




CASE MODE OF
1: (*Mode normal*)

  	ST5_5V14 := FALSE;
	ST5_5V15 := FALSE;
	ST5_5V16 := FALSE;
	
	IF ((POIDS+200) > POIDS_LIMIT) AND (GEMMA.STEP='F1' OR GEMMA.STEP='A1')  AND (PROG_STEP<100 OR PROG_STEP>=300) THEN (*Hystérésis de 200g*)
		POMPE	:= TRUE; 
	ELSIF (POIDS < POIDS_LIMIT) AND (GEMMA.STEP='F1' OR GEMMA.STEP='A1') AND (PROG_STEP<100 OR PROG_STEP>=300) THEN
		POMPE 	:= FALSE;
	ELSE
		POMPE 	:= FALSE;
	END_IF;

2:  (*Mode Vidange du réservoir d'eau*)   
    ST5_5V14 := TRUE;
	ST5_5V15 := TRUE;
	ST5_5V16 := TRUE;
	
	IF ST5_NIVEAU_EAU>2 THEN
		POMPE	:= TRUE; 
		START_TAMPO_VIDANGE := FALSE;
	ELSIF ST5_NIVEAU_EAU<0 AND NOT START_TAMPO_VIDANGE THEN
		 START_TAMPO_VIDANGE := TRUE;
	END_IF
	(*Continue de pomper encore 30 secondes depuis le niveau bas*)
	IF TAMPO_VIDANGE_TON.Q THEN
		POMPE	:= FALSE;
	END_IF
	
3:  (*Mode Remplissage du réservoir d'eau depuis le banc déminéralisateur*)   
    ST5_5V14 := FALSE;
	ST5_5V15 := TRUE;
	ST5_5V16 := FALSE;
	
	IF ST5_NIVEAU_EAU<98 THEN
		POMPE	:= TRUE; 
	ELSIF ST5_NIVEAU_EAU>100 THEN
		POMPE	:= FALSE; 
	END_IF

END_CASE;

TAMPO_VIDANGE_TON(IN:= START_TAMPO_VIDANGE, PT:=TEMPS_VIDANGE_RESERVOIR);

END_FUNCTION_BLOCK

// ---- POUs/SAFETY/SAFETY.TcPOU
PROGRAM SAFETY
VAR
END_VAR

IF SAFETY_IN.NOT_AUS_State=1 THEN

	FLAGS.SAFETY_OK:=TRUE;

ELSE

	FLAGS.SAFETY_OK:=FALSE;
END_IF;

END_PROGRAM

// ---- POUs/CONVOYER/CONVEYOR.TcPOU
PROGRAM CONVEYOR

VAR
	JIG_ST1: JIG;
	JIG_ST2: JIG;
	JIG_ST3: JIG;
	JIG_ST4: JIG;
	JIG_ST5: JIG;
	JIG_ST6: JIG;
	JIG_ST7: JIG;
	JIG_ST8: JIG;
	JIG_ST9: JIG;

	PULSE_RELEASE_JIG_OP1:TP;
	PULSE_RELEASE_JIG_OP2: TP;
	
	TEST_RELEASE :BOOL;

END_VAR
VAR_INPUT
END_VAR

(**********************************
*
* Gestion des posages Opérateur 1 et 2
*
********************************************)
IF (GEMMA.STEP='F1' OR GEMMA.STEP='F4') THEN

	(*Gestion des posages opérateur*)
	PULSE_RELEASE_JIG_OP1(IN:=(ST10_OPERATEUR1_START AND ST10_10B1) OR FLAGS.DEBUG_OPERATOR, PT:= PULSE_RELEASE_JIG_OP );
	PULSE_RELEASE_JIG_OP2(IN:=(ST10_OPERATEUR2_START AND ST10_10B2) OR FLAGS.DEBUG_OPERATOR, PT:= PULSE_RELEASE_JIG_OP );
	
	ST10_10V1:= NOT PULSE_RELEASE_JIG_OP1.Q ;
	ST10_10V2:= NOT PULSE_RELEASE_JIG_OP2.Q ;
	
	(*Activation du bon posage en fonction du débit*)
	IF ST4_5_JIG_DISABLED THEN	
		ST4_JIG_DISABLED := TRUE;
		ST5_JIG_DISABLED := TRUE;
	ELSE	
		IF PUMP_PARAMS.GEN_GRAND_DEBIT THEN
			ST4_JIG_DISABLED := TRUE;
			ST5_JIG_DISABLED := FALSE;
		ELSE
			ST4_JIG_DISABLED := FALSE;
			ST5_JIG_DISABLED := TRUE;
		END_IF
	END_IF;

END_IF;


(**********************************
*
* Gestion des posages principaux
*
********************************************)
JIG_ST1(
	CARRIER_PRESENT:=ST1_1B2 ,
	CARRIER_WAIT_PRESENT:=ST1_1B1 ,
	RELEASE_CARRIER:= FLAGS.ST1_RELEASE_CARRIER OR TEST_RELEASE,
	JIG_DISABLED:= ST1_JIG_DISABLED,
	STATUS=> FLAGS.ST1_JIG_STATUS,
	NEXT_JIG_STATUS:=JIG_ST2.STATUS,
	CYLINDER_WAIT=> ST1_1V1,
	CYLINDER_STOP=> ST1_1V3,
	CYLINDER_LOCK=> ST1_1V2);
JIG_ST2(
	CARRIER_PRESENT:=ST2_2B2 ,
	CARRIER_WAIT_PRESENT:=ST2_2B1 ,
	RELEASE_CARRIER:= FLAGS.ST2_RELEASE_CARRIER OR TEST_RELEASE,
	JIG_DISABLED:= ST2_JIG_DISABLED,
	STATUS=> FLAGS.ST2_JIG_STATUS,
	NEXT_JIG_STATUS:=JIG_ST3.STATUS,
	CYLINDER_WAIT=> ST2_2V1,
	CYLINDER_STOP=> ST2_2V3,
	CYLINDER_LOCK=> ST2_2V2);
JIG_ST3(
	CARRIER_PRESENT:=ST3_3B2 ,
	CARRIER_WAIT_PRESENT:=ST3_3B1 ,
	RELEASE_CARRIER:= FLAGS.ST3_RELEASE_CARRIER OR TEST_RELEASE,
	JIG_DISABLED:= ST3_JIG_DISABLED,
	STATUS=> FLAGS.ST3_JIG_STATUS,
	NEXT_JIG_STATUS:=JIG_ST4.STATUS,
	CYLINDER_WAIT=> ST3_3V1,
	CYLINDER_STOP=> ST3_3V3,
	CYLINDER_LOCK=> ST3_3V2);
JIG_ST4(
	CARRIER_PRESENT:=ST4_4B2 ,
	CARRIER_WAIT_PRESENT:=ST4_4B1 ,
	RELEASE_CARRIER:= FLAGS.ST4_RELEASE_CARRIER OR TEST_RELEASE,
	JIG_DISABLED:= ST4_JIG_DISABLED,
	STATUS=> FLAGS.ST4_JIG_STATUS,
	NEXT_JIG_STATUS:=JIG_ST5.STATUS,
	CYLINDER_WAIT=> ST4_4V1,
	CYLINDER_STOP=> ST4_4V3,
	CYLINDER_LOCK=> ST4_4V2);
JIG_ST5(
	CARRIER_PRESENT:=ST5_5B2 ,
	CARRIER_WAIT_PRESENT:=ST5_5B1 ,
	RELEASE_CARRIER:= FLAGS.ST5_RELEASE_CARRIER OR TEST_RELEASE,
	JIG_DISABLED:= ST5_JIG_DISABLED,
	STATUS=> FLAGS.ST5_JIG_STATUS,
	NEXT_JIG_STATUS:=JIG_ST6.STATUS,
	CYLINDER_WAIT=> ST5_5V1,
	CYLINDER_STOP=> ST5_5V3,
	CYLINDER_LOCK=> ST5_5V2);
JIG_ST6(
	CARRIER_PRESENT:=ST6_6B2 ,
	CARRIER_WAIT_PRESENT:=ST6_6B1 ,
	RELEASE_CARRIER:= FLAGS.ST6_RELEASE_CARRIER OR TEST_RELEASE,
	JIG_DISABLED:= ST6_JIG_DISABLED,
	STATUS=> FLAGS.ST6_JIG_STATUS,
	NEXT_JIG_STATUS:=JIG_ST7.STATUS,
	CYLINDER_WAIT=> ST6_6V1,
	CYLINDER_STOP=> ST6_6V3,
	CYLINDER_LOCK=> ST6_6V2);
JIG_ST7(
	CARRIER_PRESENT:=ST7_7B2 ,
	CARRIER_WAIT_PRESENT:=ST7_7B1 ,
	RELEASE_CARRIER:= FLAGS.ST7_RELEASE_CARRIER OR TEST_RELEASE,
	JIG_DISABLED:= ST7_JIG_DISABLED,
	STATUS=> FLAGS.ST7_JIG_STATUS,
	NEXT_JIG_STATUS:=JIG_ST8.STATUS,
	CYLINDER_WAIT=> ST7_7V1,
	CYLINDER_STOP=> ST7_7V3,
	CYLINDER_LOCK=> ST7_7V2);
JIG_ST8(
	CARRIER_PRESENT:=ST8_8B2 ,
	CARRIER_WAIT_PRESENT:=ST8_8B1 ,
	RELEASE_CARRIER:= FLAGS.ST8_RELEASE_CARRIER OR TEST_RELEASE,
	JIG_DISABLED:= ST8_JIG_DISABLED,
	STATUS=> FLAGS.ST8_JIG_STATUS,
	NEXT_JIG_STATUS:=JIG_ST9.STATUS,
	CYLINDER_WAIT=> ST8_8V1,
	CYLINDER_STOP=> ST8_8V3,
	CYLINDER_LOCK=> ST8_8V2);	
JIG_ST9(
	CARRIER_PRESENT:=ST9_9B2 ,
	CARRIER_WAIT_PRESENT:=ST9_9B1 ,
	RELEASE_CARRIER:= FLAGS.ST9_RELEASE_CARRIER OR TEST_RELEASE,
	JIG_DISABLED:= ST9_JIG_DISABLED,
	STATUS=> FLAGS.ST9_JIG_STATUS,
	NEXT_JIG_STATUS:=FALSE,
	CYLINDER_WAIT=> ST9_9V1,
	CYLINDER_STOP=> ST9_9V3,
	CYLINDER_LOCK=> ST9_9V2);

END_PROGRAM

// ---- POUs/CONVOYER/JIG.TcPOU
FUNCTION_BLOCK JIG
VAR
	STEP: INT := 0; (* Internal program step *)
	TIMER_RELEASE: TON;
	START_RELEASE_TIMER:BOOL:=FALSE;
END_VAR

VAR_INPUT
	NEXT_JIG_STATUS:BOOL; (*Status of the next jig*)
	CARRIER_PRESENT:BOOL; (*CARRIER IS PRESENT *)
	CARRIER_WAIT_PRESENT:BOOL; (*CARRIER IS PRESENT *)
	RELEASE_CARRIER:BOOL; (*Ask the function to release the carrier *)
	JIG_DISABLED: BOOL; (*Disable the JIG *)
END_VAR

VAR_OUTPUT
	STATUS: BOOL := FALSE; (* 0-> JIG FREE   1-> JIB BUSY *)
	CYLINDER_STOP: BOOL :=FALSE; (* STOP the carrier at this position *)
	CYLINDER_LOCK: BOOL:=FALSE; (* LOCK the carrier at this position *)
	CYLINDER_WAIT: BOOL:=FALSE; (* vérin pour bloquer les palettes avant le poste*)
END_VAR

(************************************************************************************************************************************
*
* Gère le posage principale pour une station (Palette et convoyeur)
*
*
************************************************************************************************************************************)
IF GEMMA.STEP='A6' OR GEMMA.STEP='D1' OR JIG_DISABLED THEN
	STEP:=0;
END_IF;

CASE STEP OF

0: (*Init*)
	STEP:=STEP+1;
	STATUS:=0;
	START_RELEASE_TIMER:=FALSE;
	CYLINDER_STOP:=FALSE;
	CYLINDER_LOCK:=FALSE;
	CYLINDER_WAIT:=FALSE;

1: (*Wait for a carrier*)
	CYLINDER_STOP:=TRUE;
	
	IF CARRIER_PRESENT THEN
		CYLINDER_LOCK:=TRUE;
		CYLINDER_WAIT:=TRUE;
		STATUS:=1;
		STEP:=STEP+1;
	END_IF;
	IF CARRIER_WAIT_PRESENT AND CARRIER_PRESENT THEN (*Lock a carrier behind only if a carrier is already locked at the working position*)
		CYLINDER_WAIT:=TRUE;
	END_IF
	

2: (*Release the carrier*)
	
	IF RELEASE_CARRIER AND NEXT_JIG_STATUS=0 THEN
		CYLINDER_LOCK:=FALSE;
		CYLINDER_STOP:=FALSE;
		CYLINDER_WAIT:=FALSE;
		START_RELEASE_TIMER:=1;
		STEP:=STEP+1;
	END_IF;

3: (*Delay after release of the carrier*)
	IF TIMER_RELEASE.Q THEN
		CYLINDER_LOCK:=FALSE;
		CYLINDER_STOP:=FALSE;
		CYLINDER_WAIT:=FALSE;
		START_RELEASE_TIMER:=0;
		STATUS:=0;
		STEP:=1;
	END_IF;







ELSE
    ;
END_CASE;


(* TIMERS*)
TIMER_RELEASE(IN:=START_RELEASE_TIMER,PT:=CARRIER_RELEASE_DELAY);

END_FUNCTION_BLOCK

// ---- POUs/AIs/AIS.TcPOU
PROGRAM AIS
VAR
	ST2_2P1_CONVERT: WIKA_GET_VALUES;
	ST4_4P1_CONVERT: WIKA_GET_VALUES;
	ST4_4P2_CONVERT: WIKA_GET_VALUES;
	ST5_5P1_CONVERT: WIKA_GET_VALUES;
	ST5_5P2_CONVERT: WIKA_GET_VALUES;
	ST6_6P1_CONVERT: WIKA_GET_VALUES;
	ST4_GetPositionIs: FB_GetPositionIs;
	ST5_GetPositionIs: FB_GetPositionIs;
	
	FB_CTRL_PT3_ST4_PRESSURE: FB_CTRL_PT3;
	FB_CTRL_PT3_ST5_PRESSURE: FB_CTRL_PT3;
	eMode_PRESSION: E_CTRL_MODE;
	stParams_PRESSION: ST_CTRL_PT3_PARAMS;
END_VAR

(**********************************************************************
*
*Conversion des entrées analogiques
*
*
*************************************************************************)



(*STATION 1***************************************************************************)
ST2_2P1_CONVERT(
INPUTS:= ST2_2P1.VALUE, 
Pressure=> ST2_VACUUM,);

(*STATION 3***************************************************************************)
ST3_PRESSION := ST3_3P1/32768.0*10; (*32768 pour 16 bits bipolair et 10 pour 10mBar*)
ST3_PRESSION_ABS := ST3_3P2/32768.0*100000; (*32768 pour 16 bits bipolair et 10 pour 10mBar*)

(*STATION 4***************************************************************************)
ST4_4P1_CONVERT(
INPUTS:= ST4_4P1.VALUE, 
Pressure=> ST4_VACUUM,);

ST4_4P2_CONVERT(
INPUTS:= ST4_4P2.VALUE, 
Pressure=> ST4_PRESSURE,);

(*Filtres 3 ème ordre*)
FB_CTRL_PT3_ST4_PRESSURE(
	fIn:= ST4_PRESSURE,
	fManValue:= 0,
	eMode:= eMode_PRESSION,
	bHold:= FALSE ,
	stParams:= stParams_PRESSION,
	fOut=> ST4_PRESSURE_FILTERED );

ST4_COURANT:=ST4_Multimeter_value/1000.0;

ST4_GetPositionIs(
	ADSNetId:= MOTOR_ST4_ADDRESS, 
	NodeId:= 1, 
	Read:= TRUE, 
	PositionIs=> FLAGS.MOTOR_ST4_ACTUAL_POSITION);

(*STATION 5***************************************************************************)
ST5_5P1_CONVERT(
INPUTS:= ST5_5P1.VALUE, 
Pressure=> ST5_VACUUM,);

ST5_5P2_CONVERT(
INPUTS:= ST5_5P2.VALUE, 
Pressure=> ST5_PRESSURE,);

(*Filtres 3 ème ordre*)
FB_CTRL_PT3_ST5_PRESSURE(
	fIn:= ST5_PRESSURE,
	fManValue:= 0,
	eMode:= eMode_PRESSION,
	bHold:= FALSE ,
	stParams:= stParams_PRESSION,
	fOut=> ST5_PRESSURE_FILTERED );

ST5_COURANT:=ST5_Multimeter_value/1000.0;

ST5_GetPositionIs(
	ADSNetId:= MOTOR_ST4_ADDRESS, 
	NodeId:= 1, 
	Read:= TRUE, 
	PositionIs=> FLAGS.MOTOR_ST5_ACTUAL_POSITION);
	
ST5_NIVEAU_EAU := ST5_Niveau_Reservoir * 100 /(RESERVOIR_EAU_MAX-RESERVOIR_EAU_MIN) + 100*RESERVOIR_EAU_MIN/(RESERVOIR_EAU_MIN-RESERVOIR_EAU_MAX);

(*STATION 6***************************************************************************)
ST6_6P1_CONVERT(
INPUTS:= ST6_6P1.VALUE, 
Pressure=> ST6_PRESSURE,);

(*PARAMETRES FILTRES*********************************************************************)

(* init parameter struct *)
stParams_PRESSION.tCtrlCycleTime		:= T#10MS;
stParams_PRESSION.tTaskCycleTime		:= T#10MS;
stParams_PRESSION.tT1					:= T#600MS;
stParams_PRESSION.tT2					:= T#600MS;
stParams_PRESSION.tT3					:= T#600MS;
stParams_PRESSION.fKp					:= 1;

(* set the mode to ACTIVE --> normal operation *)
eMode_PRESSION							:= eCTRL_MODE_ACTIVE;

END_PROGRAM

// ---- POUs/WIKA/WIKA_GET_VALUES.TcPOU
FUNCTION_BLOCK WIKA_GET_VALUES

VAR_INPUT
	INPUTS: ARRAY [0..7] OF USINT;
END_VAR

VAR_OUTPUT
	Pressure: REAL;
	Measuring_Type:BOOL; (*0->Relativ 1->Absolute*)
END_VAR

VAR
	Pressure_Value:REAL;
	Sign:SINT;
	Sign_Exponent:INT;
	Exponent:REAL;
END_VAR

Pressure_Value:= 	BOOL_TO_INT(INPUTS[1].0)*1 +
			BOOL_TO_INT(INPUTS[1].1)*2 +
			BOOL_TO_INT(INPUTS[1].2)*4 +
			BOOL_TO_INT(INPUTS[1].3)*8 +
			BOOL_TO_INT(INPUTS[1].4)*16 +
			BOOL_TO_INT(INPUTS[1].5)*32 +
			BOOL_TO_INT(INPUTS[1].6)*64 +
			BOOL_TO_INT(INPUTS[1].7)*128+
			BOOL_TO_INT(INPUTS[0].0)*256 +
			BOOL_TO_INT(INPUTS[0].1)*512 +
			BOOL_TO_INT(INPUTS[0].2)*1024 +
			BOOL_TO_INT(INPUTS[0].3)*2048 +
			BOOL_TO_INT(INPUTS[0].4)*4096 +
			BOOL_TO_INT(INPUTS[0].5)*8192 +
			BOOL_TO_INT(INPUTS[0].6)*16384;

IF INPUTS[0].7=0 THEN
Sign:=1;
ELSE
Sign:=-1;
END_IF

Measuring_Type:=INPUTS[2].7;

Sign_Exponent:=BOOL_TO_SINT(INPUTS[2].6)*-1;

Exponent:=	EXPT(10,(BOOL_TO_INT(INPUTS[2].3)*1 + BOOL_TO_INT(INPUTS[2].4)*2 + BOOL_TO_INT(INPUTS[2].5)*4)*Sign_Exponent);

Pressure:=Exponent*Pressure_Value*Sign;

END_FUNCTION_BLOCK

// ---- POUs/AIs/ST45_TO_HMI.TcPOU
PROGRAM ST45_TO_HMI
VAR
END_VAR

IF PUMP_PARAMS.GEN_GRAND_DEBIT THEN
	
	ST45_QMAX			:=	ST5_QMAX;
	ST45_Q				:=	ST5_Q;
	ST45_PRESSURE		:=	ST5_PRESSURE_FILTERED;
	ST45_VACUUM			:=	ST5_VACUUM;
	ST45_POIDS			:=	ST5_POIDS;
	
	ST45_COURANT		:=	ST5_COURANT;
	
ELSE
	
	ST45_QMAX			:=	ST4_QMAX;
	ST45_Q				:=	ST4_Q;
	ST45_PRESSURE		:=	ST4_PRESSURE_FILTERED;
	ST45_VACUUM			:=	ST4_VACUUM;
	ST45_POIDS			:=	ST4_POIDS;
	
	ST45_COURANT		:=	ST4_COURANT;
	
END_IF

END_PROGRAM

// ---- POUs/MAXON/ST4_MOTOR.TcPOU
PROGRAM ST4_MOTOR
VAR
	ClearFault: FB_ClearFault;
	SetEnableState: FB_SetEnableState;
	SetHomingParameter: FB_SetHomingParameter;
	FindHome: FB_FindHome;
	POSITION: DINT;
	GetMovementState: FB_GetMovementState;
	MoveToPosition: FB_MoveToPosition;
	SetOperationMode: FB_SetOperationMode;
	SetMotorParameter: FB_SetMotorParameter;
	SetPositionProfile: FB_SetPositionProfile;
END_VAR

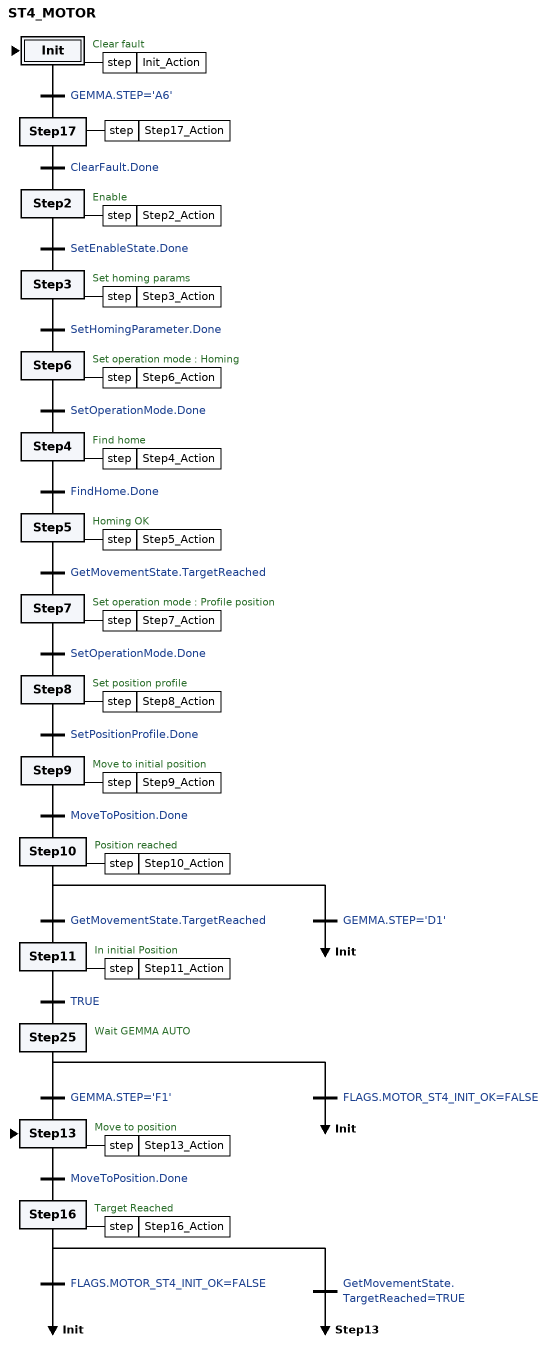
// Clear fault
INITIAL_STEP Init:
    Init_Action(N);  // step action
END_STEP
TRANSITION FROM Init TO Step17
    := GEMMA.STEP='A6';
END_TRANSITION
STEP Step17:
    Step17_Action(N);  // step action
END_STEP
TRANSITION FROM Step17 TO Step2
    := ClearFault.Done;
END_TRANSITION
// Enable
STEP Step2:
    Step2_Action(N);  // step action
END_STEP
TRANSITION FROM Step2 TO Step3
    := SetEnableState.Done;
END_TRANSITION
// Set homing params
STEP Step3:
    Step3_Action(N);  // step action
END_STEP
TRANSITION FROM Step3 TO Step6
    := SetHomingParameter.Done;
END_TRANSITION
// Set operation mode : Homing
STEP Step6:
    Step6_Action(N);  // step action
END_STEP
TRANSITION FROM Step6 TO Step4
    := SetOperationMode.Done;
END_TRANSITION
// Find home
STEP Step4:
    Step4_Action(N);  // step action
END_STEP
TRANSITION FROM Step4 TO Step5
    := FindHome.Done;
END_TRANSITION
// Homing OK
STEP Step5:
    Step5_Action(N);  // step action
END_STEP
TRANSITION FROM Step5 TO Step7
    := GetMovementState.TargetReached;
END_TRANSITION
// Set operation mode : Profile position
STEP Step7:
    Step7_Action(N);  // step action
END_STEP
TRANSITION FROM Step7 TO Step8
    := SetOperationMode.Done;
END_TRANSITION
// Set position profile
STEP Step8:
    Step8_Action(N);  // step action
END_STEP
TRANSITION FROM Step8 TO Step9
    := SetPositionProfile.Done;
END_TRANSITION
// Move to initial position
STEP Step9:
    Step9_Action(N);  // step action
END_STEP
TRANSITION FROM Step9 TO Step10
    := MoveToPosition.Done;
END_TRANSITION
// Position reached
STEP Step10:
    Step10_Action(N);  // step action
END_STEP
TRANSITION FROM Step10 TO Step11
    := GetMovementState.TargetReached;
END_TRANSITION
TRANSITION FROM Step10 TO Init
    := GEMMA.STEP='D1';
END_TRANSITION
// In initial Position
STEP Step11:
    Step11_Action(N);  // step action
END_STEP
TRANSITION FROM Step11 TO Step25
    := TRUE;
END_TRANSITION
// Wait GEMMA AUTO
STEP Step25:
END_STEP
TRANSITION FROM Step25 TO Step13
    := GEMMA.STEP='F1';
END_TRANSITION
TRANSITION FROM Step25 TO Init
    := FLAGS.MOTOR_ST4_INIT_OK=FALSE;
END_TRANSITION
// Move to position
STEP Step13:
    Step13_Action(N);  // step action
END_STEP
TRANSITION FROM Step13 TO Step16
    := MoveToPosition.Done;
END_TRANSITION
// Target Reached
STEP Step16:
    Step16_Action(N);  // step action
END_STEP
TRANSITION FROM Step16 TO Init
    := FLAGS.MOTOR_ST4_INIT_OK=FALSE;
END_TRANSITION
TRANSITION FROM Step16 TO Step13
    := GetMovementState.TargetReached=TRUE;
END_TRANSITION

ACTION Step5_Action:
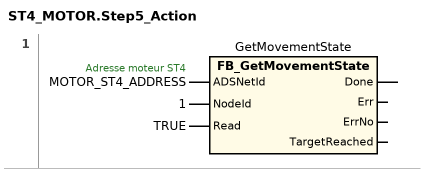
// NETWORK 1
//   MOTOR_ST4_ADDRESS: Adresse moteur ST4
GetMovementState(ADSNetId := MOTOR_ST4_ADDRESS, NodeId := 1, Read := TRUE); // FB_GetMovementState
END_ACTION

ACTION Step16_Action:
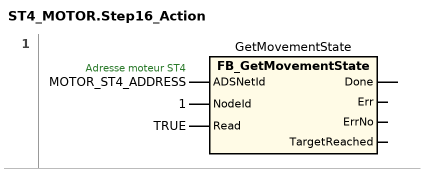
// NETWORK 1
//   MOTOR_ST4_ADDRESS: Adresse moteur ST4
GetMovementState(ADSNetId := MOTOR_ST4_ADDRESS, NodeId := 1, Read := TRUE); // FB_GetMovementState
END_ACTION

ACTION Step7_Action:
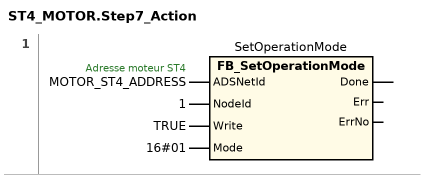
// NETWORK 1
//   MOTOR_ST4_ADDRESS: Adresse moteur ST4
SetOperationMode(ADSNetId := MOTOR_ST4_ADDRESS, NodeId := 1, Write := TRUE, Mode := 16#01); // FB_SetOperationMode
END_ACTION

ACTION Step2_Action:
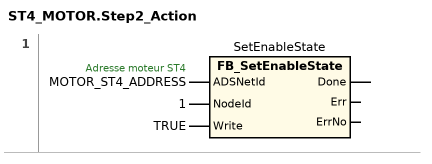
// NETWORK 1
//   MOTOR_ST4_ADDRESS: Adresse moteur ST4
SetEnableState(ADSNetId := MOTOR_ST4_ADDRESS, NodeId := 1, Write := TRUE); // FB_SetEnableState
END_ACTION

ACTION Step17_Action:
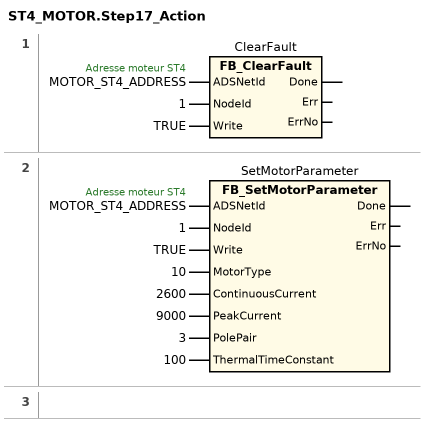
// NETWORK 1
//   MOTOR_ST4_ADDRESS: Adresse moteur ST4
ClearFault(ADSNetId := MOTOR_ST4_ADDRESS, NodeId := 1, Write := TRUE); // FB_ClearFault

// NETWORK 2
//   MOTOR_ST4_ADDRESS: Adresse moteur ST4
SetMotorParameter(
    ADSNetId := MOTOR_ST4_ADDRESS,
    NodeId := 1,
    Write := TRUE,
    MotorType := 10,
    ContinuousCurrent := 2600,
    PeakCurrent := 9000,
    PolePair := 3,
    ThermalTimeConstant := 100); // FB_SetMotorParameter

// NETWORK 3
END_ACTION

ACTION Step6_Action:
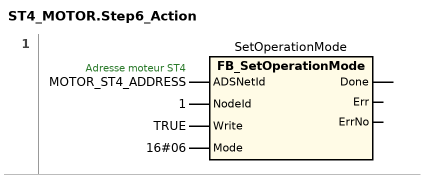
// NETWORK 1
//   MOTOR_ST4_ADDRESS: Adresse moteur ST4
SetOperationMode(ADSNetId := MOTOR_ST4_ADDRESS, NodeId := 1, Write := TRUE, Mode := 16#06); // FB_SetOperationMode
END_ACTION

ACTION Step13_Action:
(*Limitation deplacement Moteur*)
(*IF FLAGS.MOTOR_ST4_POSITION>MOTOR_ST4_POSITION_MAX THEN
	POSITION:=MOTOR_ST4_POSITION_MAX;
ELSIF FLAGS.MOTOR_ST4_POSITION<0 THEN
	POSITION:=0;
ELSE
	POSITION:=FLAGS.MOTOR_ST4_POSITION;
END_IF*)

POSITION:=FLAGS.MOTOR_ST4_POSITION;

MoveToPosition(
	ADSNetId:= MOTOR_ST4_ADDRESS,
	NodeId:= 1,
	Write:= TRUE,
	TargetPosition:= POSITION,
	Absolut:= TRUE);
END_ACTION

ACTION Step10_Action:
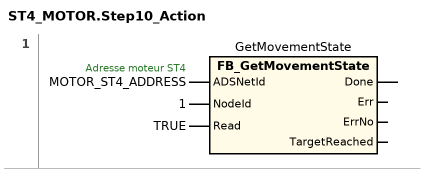
// NETWORK 1
//   MOTOR_ST4_ADDRESS: Adresse moteur ST4
GetMovementState(ADSNetId := MOTOR_ST4_ADDRESS, NodeId := 1, Read := TRUE); // FB_GetMovementState
END_ACTION

ACTION Step3_Action:
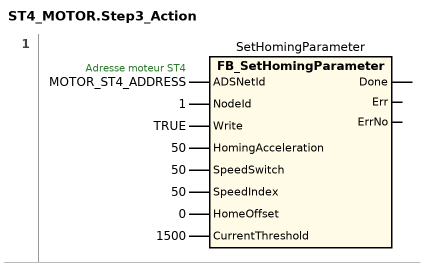
// NETWORK 1
//   MOTOR_ST4_ADDRESS: Adresse moteur ST4
SetHomingParameter(
    ADSNetId := MOTOR_ST4_ADDRESS,
    NodeId := 1,
    Write := TRUE,
    HomingAcceleration := 50,
    SpeedSwitch := 50,
    SpeedIndex := 50,
    HomeOffset := 0,
    CurrentThreshold := 1500); // FB_SetHomingParameter
END_ACTION

ACTION Step9_Action:
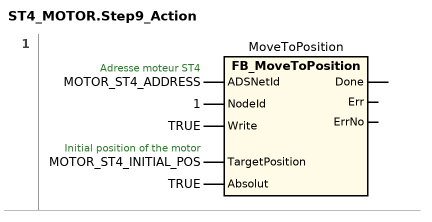
// NETWORK 1
//   MOTOR_ST4_ADDRESS: Adresse moteur ST4
//   MOTOR_ST4_INITIAL_POS: Initial position of the motor
MoveToPosition(
    ADSNetId := MOTOR_ST4_ADDRESS,
    NodeId := 1,
    Write := TRUE,
    TargetPosition := MOTOR_ST4_INITIAL_POS,
    Absolut := TRUE); // FB_MoveToPosition
END_ACTION

ACTION Step8_Action:
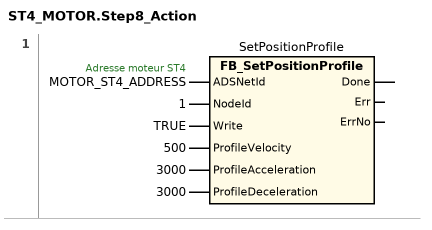
// NETWORK 1
//   MOTOR_ST4_ADDRESS: Adresse moteur ST4
SetPositionProfile(
    ADSNetId := MOTOR_ST4_ADDRESS,
    NodeId := 1,
    Write := TRUE,
    ProfileVelocity := 500,
    ProfileAcceleration := 3000,
    ProfileDeceleration := 3000); // FB_SetPositionProfile
END_ACTION

ACTION Step11_Action:

(*SetDisableState(
	ADSNetId:= '10.0.0.31.6.1',
	NodeId:= 1,
	Write:= TRUE);*)

FLAGS.MOTOR_ST4_INIT_OK:=TRUE;
END_ACTION

ACTION Init_Action:

END_ACTION

ACTION Step4_Action:
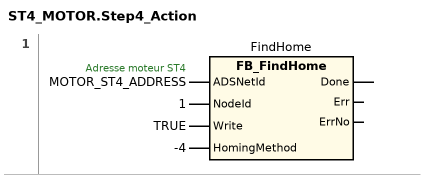
// NETWORK 1
//   MOTOR_ST4_ADDRESS: Adresse moteur ST4
FindHome(ADSNetId := MOTOR_ST4_ADDRESS, NodeId := 1, Write := TRUE, HomingMethod := -4); // FB_FindHome
END_ACTION

END_PROGRAM

// ---- POUs/MAXON/ST5_MOTOR.TcPOU
PROGRAM ST5_MOTOR
VAR
	ClearFault: FB_ClearFault;
	SetEnableState: FB_SetEnableState;
	SetHomingParameter: FB_SetHomingParameter;
	FindHome: FB_FindHome;
	POSITION: DINT;
	GetMovementState: FB_GetMovementState;
	MoveToPosition: FB_MoveToPosition;
	SetOperationMode: FB_SetOperationMode;
	SetMotorParameter: FB_SetMotorParameter;
	SetPositionProfile: FB_SetPositionProfile;
END_VAR

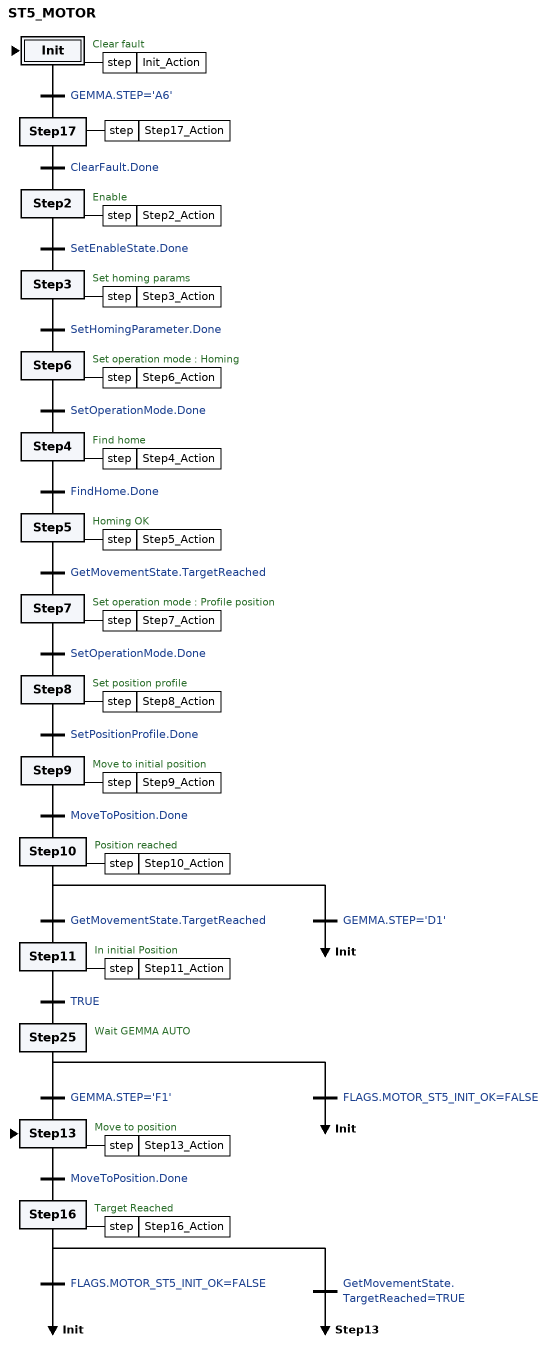
// Clear fault
INITIAL_STEP Init:
    Init_Action(N);  // step action
END_STEP
TRANSITION FROM Init TO Step17
    := GEMMA.STEP='A6';
END_TRANSITION
STEP Step17:
    Step17_Action(N);  // step action
END_STEP
TRANSITION FROM Step17 TO Step2
    := ClearFault.Done;
END_TRANSITION
// Enable
STEP Step2:
    Step2_Action(N);  // step action
END_STEP
TRANSITION FROM Step2 TO Step3
    := SetEnableState.Done;
END_TRANSITION
// Set homing params
STEP Step3:
    Step3_Action(N);  // step action
END_STEP
TRANSITION FROM Step3 TO Step6
    := SetHomingParameter.Done;
END_TRANSITION
// Set operation mode : Homing
STEP Step6:
    Step6_Action(N);  // step action
END_STEP
TRANSITION FROM Step6 TO Step4
    := SetOperationMode.Done;
END_TRANSITION
// Find home
STEP Step4:
    Step4_Action(N);  // step action
END_STEP
TRANSITION FROM Step4 TO Step5
    := FindHome.Done;
END_TRANSITION
// Homing OK
STEP Step5:
    Step5_Action(N);  // step action
END_STEP
TRANSITION FROM Step5 TO Step7
    := GetMovementState.TargetReached;
END_TRANSITION
// Set operation mode : Profile position
STEP Step7:
    Step7_Action(N);  // step action
END_STEP
TRANSITION FROM Step7 TO Step8
    := SetOperationMode.Done;
END_TRANSITION
// Set position profile
STEP Step8:
    Step8_Action(N);  // step action
END_STEP
TRANSITION FROM Step8 TO Step9
    := SetPositionProfile.Done;
END_TRANSITION
// Move to initial position
STEP Step9:
    Step9_Action(N);  // step action
END_STEP
TRANSITION FROM Step9 TO Step10
    := MoveToPosition.Done;
END_TRANSITION
// Position reached
STEP Step10:
    Step10_Action(N);  // step action
END_STEP
TRANSITION FROM Step10 TO Step11
    := GetMovementState.TargetReached;
END_TRANSITION
TRANSITION FROM Step10 TO Init
    := GEMMA.STEP='D1';
END_TRANSITION
// In initial Position
STEP Step11:
    Step11_Action(N);  // step action
END_STEP
TRANSITION FROM Step11 TO Step25
    := TRUE;
END_TRANSITION
// Wait GEMMA AUTO
STEP Step25:
END_STEP
TRANSITION FROM Step25 TO Step13
    := GEMMA.STEP='F1';
END_TRANSITION
TRANSITION FROM Step25 TO Init
    := FLAGS.MOTOR_ST5_INIT_OK=FALSE;
END_TRANSITION
// Move to position
STEP Step13:
    Step13_Action(N);  // step action
END_STEP
TRANSITION FROM Step13 TO Step16
    := MoveToPosition.Done;
END_TRANSITION
// Target Reached
STEP Step16:
    Step16_Action(N);  // step action
END_STEP
TRANSITION FROM Step16 TO Init
    := FLAGS.MOTOR_ST5_INIT_OK=FALSE;
END_TRANSITION
TRANSITION FROM Step16 TO Step13
    := GetMovementState.TargetReached=TRUE;
END_TRANSITION

ACTION Step2_Action:
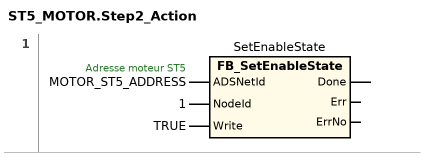
// NETWORK 1
//   MOTOR_ST5_ADDRESS: Adresse moteur ST5
SetEnableState(ADSNetId := MOTOR_ST5_ADDRESS, NodeId := 1, Write := TRUE); // FB_SetEnableState
END_ACTION

ACTION Step16_Action:
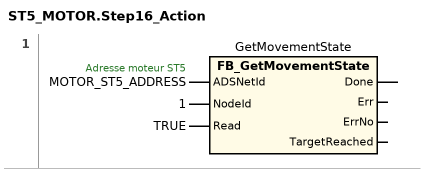
// NETWORK 1
//   MOTOR_ST5_ADDRESS: Adresse moteur ST5
GetMovementState(ADSNetId := MOTOR_ST5_ADDRESS, NodeId := 1, Read := TRUE); // FB_GetMovementState
END_ACTION

ACTION Step13_Action:
(*Limitation deplacement Moteur*)
IF FLAGS.MOTOR_ST5_POSITION>MOTOR_ST5_POSITION_MAX THEN
	POSITION:=MOTOR_ST5_POSITION_MAX;
ELSIF FLAGS.MOTOR_ST5_POSITION<0 THEN
	POSITION:=0;
ELSE
	POSITION:=FLAGS.MOTOR_ST5_POSITION;
END_IF


MoveToPosition(
	ADSNetId:= MOTOR_ST5_ADDRESS,
	NodeId:= 1,
	Write:= TRUE,
	TargetPosition:= POSITION,
	Absolut:= TRUE);
END_ACTION

ACTION Step5_Action:
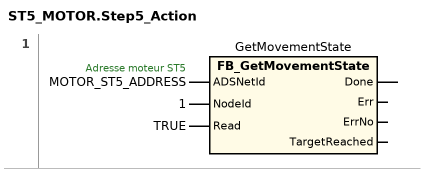
// NETWORK 1
//   MOTOR_ST5_ADDRESS: Adresse moteur ST5
GetMovementState(ADSNetId := MOTOR_ST5_ADDRESS, NodeId := 1, Read := TRUE); // FB_GetMovementState
END_ACTION

ACTION Step10_Action:
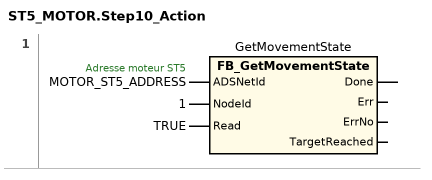
// NETWORK 1
//   MOTOR_ST5_ADDRESS: Adresse moteur ST5
GetMovementState(ADSNetId := MOTOR_ST5_ADDRESS, NodeId := 1, Read := TRUE); // FB_GetMovementState
END_ACTION

ACTION Step9_Action:
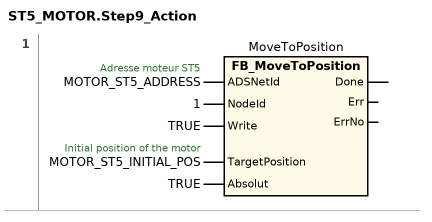
// NETWORK 1
//   MOTOR_ST5_ADDRESS: Adresse moteur ST5
//   MOTOR_ST5_INITIAL_POS: Initial position of the motor
MoveToPosition(
    ADSNetId := MOTOR_ST5_ADDRESS,
    NodeId := 1,
    Write := TRUE,
    TargetPosition := MOTOR_ST5_INITIAL_POS,
    Absolut := TRUE); // FB_MoveToPosition
END_ACTION

ACTION Step11_Action:

(*SetDisableState(
	ADSNetId:= '10.0.0.31.6.1',
	NodeId:= 1,
	Write:= TRUE);*)

FLAGS.MOTOR_ST5_INIT_OK:=TRUE;
END_ACTION

ACTION Step8_Action:
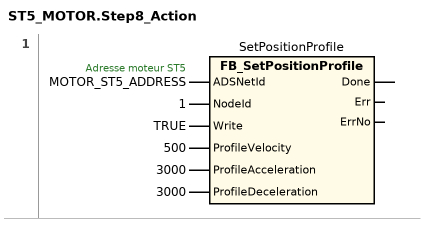
// NETWORK 1
//   MOTOR_ST5_ADDRESS: Adresse moteur ST5
SetPositionProfile(
    ADSNetId := MOTOR_ST5_ADDRESS,
    NodeId := 1,
    Write := TRUE,
    ProfileVelocity := 500,
    ProfileAcceleration := 3000,
    ProfileDeceleration := 3000); // FB_SetPositionProfile
END_ACTION

ACTION Step6_Action:
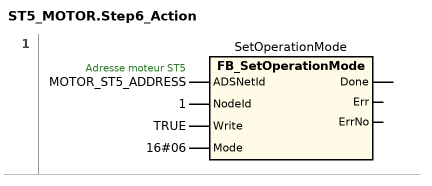
// NETWORK 1
//   MOTOR_ST5_ADDRESS: Adresse moteur ST5
SetOperationMode(ADSNetId := MOTOR_ST5_ADDRESS, NodeId := 1, Write := TRUE, Mode := 16#06); // FB_SetOperationMode
END_ACTION

ACTION Init_Action:

END_ACTION

ACTION Step3_Action:
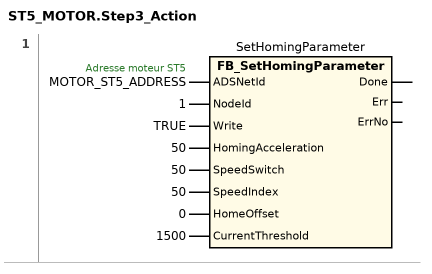
// NETWORK 1
//   MOTOR_ST5_ADDRESS: Adresse moteur ST5
SetHomingParameter(
    ADSNetId := MOTOR_ST5_ADDRESS,
    NodeId := 1,
    Write := TRUE,
    HomingAcceleration := 50,
    SpeedSwitch := 50,
    SpeedIndex := 50,
    HomeOffset := 0,
    CurrentThreshold := 1500); // FB_SetHomingParameter
END_ACTION

ACTION Step17_Action:
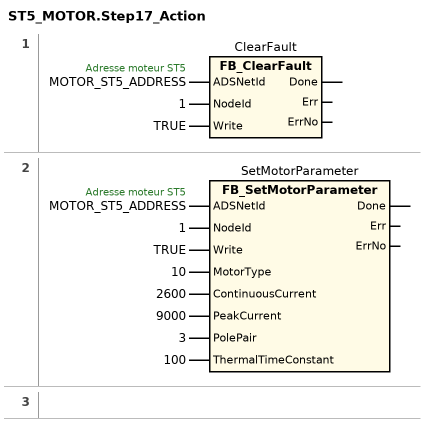
// NETWORK 1
//   MOTOR_ST5_ADDRESS: Adresse moteur ST5
ClearFault(ADSNetId := MOTOR_ST5_ADDRESS, NodeId := 1, Write := TRUE); // FB_ClearFault

// NETWORK 2
//   MOTOR_ST5_ADDRESS: Adresse moteur ST5
SetMotorParameter(
    ADSNetId := MOTOR_ST5_ADDRESS,
    NodeId := 1,
    Write := TRUE,
    MotorType := 10,
    ContinuousCurrent := 2600,
    PeakCurrent := 9000,
    PolePair := 3,
    ThermalTimeConstant := 100); // FB_SetMotorParameter

// NETWORK 3
END_ACTION

ACTION Step4_Action:
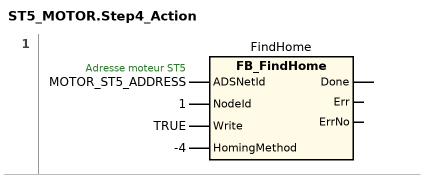
// NETWORK 1
//   MOTOR_ST5_ADDRESS: Adresse moteur ST5
FindHome(ADSNetId := MOTOR_ST5_ADDRESS, NodeId := 1, Write := TRUE, HomingMethod := -4); // FB_FindHome
END_ACTION

ACTION Step7_Action:
